FUNCTION "LAnyAxis_UnpubPhasingRelativeMasterProxy" : Void   // FC30054, SCL
TITLE = LAnyAxis_UnpubPhasingRelativeMasterProxy
{ S7_Optimized_Access := 'TRUE' }
AUTHOR : tech.team.motioncontrol@siemens.com
FAMILY : AnyAxis
VERSION : 1.0
// Support: tech.team.motioncontrol@siemens.com
   VAR_INPUT
      slave : TO_SynchronousAxis;   // Slave axis specification
      master : TO_LeadingAxisProxy;   // Master axis specification
   END_VAR
   VAR_IN_OUT
      instMC : MC_PHASINGRELATIVE;   // Instance of MC_Instruction
   END_VAR
   // Ret_Val : No return value
BEGIN
   // Call of MC_Instruction
   #instMC(Master := #master,
           Slave := #slave);
END_FUNCTION

FUNCTION "LAnyAxis_UnpubPhasingRelativeMasterSyncAxis" : Void   // FC30055, SCL
TITLE = LAnyAxis_UnpubPhasingRelativeMasterSyncAxis
{ S7_Optimized_Access := 'TRUE' }
AUTHOR : tech.team.motioncontrol@siemens.com
FAMILY : AnyAxis
VERSION : 1.0
// Support: tech.team.motioncontrol@siemens.com
   VAR_INPUT
      slave : TO_SynchronousAxis;   // Slave axis specification
      master : TO_SynchronousAxis;   // Master axis specification
   END_VAR
   VAR_IN_OUT
      instMC : MC_PHASINGRELATIVE;   // Instance of MC_Instruction
   END_VAR
   // Ret_Val : No return value
BEGIN
   // Call of MC_Instruction
   #instMC(Master := #master,
           Slave := #slave);
END_FUNCTION

// folder: LAnyAxis_Blocks/LAnyAxis_MC_TorqueData

FUNCTION_BLOCK "LAnyAxis_MC_TorqueLimiting"   // FB30042, SCL
TITLE = LAnyAxis_MC_TorqueLimiting
{ S7_Optimized_Access := 'TRUE' }
AUTHOR : tech.team.motioncontrol@siemens.com
FAMILY : AnyAxis
VERSION : 1.0
// Support: tech.team.motioncontrol@siemens.com 
// See corresponding MC_ instruction in TIA Portal help (information system)
   VAR_INPUT
      Axis : DB_ANY;   // See corresponding parameter of MC_ instruction in TIA Portal help (information system)
      Enable : Bool;   // See corresponding parameter of MC_ instruction in TIA Portal help (information system)
      Limit : LReal := -1.0;   // See corresponding parameter of MC_ instruction in TIA Portal help (information system)
      Mode : DInt;   // See corresponding parameter of MC_ instruction in TIA Portal help (information system)
   END_VAR
   VAR_OUTPUT
      InClamping : Bool;   // See corresponding parameter of MC_ instruction in TIA Portal help (information system)
      InLimitation : Bool;   // See corresponding parameter of MC_ instruction in TIA Portal help (information system)
      Busy : Bool;   // See corresponding parameter of MC_ instruction in TIA Portal help (information system)
      Error : Bool;   // See corresponding parameter of MC_ instruction in TIA Portal help (information system)
      ErrorId : Word;   // See corresponding parameter of MC_ instruction in TIA Portal help (information system)
   END_VAR
   VAR
      instMC : MC_TORQUELIMITING;   // Instance of MC_Instruction
      statEnableOld : Bool;   // Old value of execute
      statAxis : DB_ANY;   // Internal variable of axis
      statAxisType : Int;   // Actual state / axis type
   END_VAR
   VAR CONSTANT
      ERROR_INVALID_TECHNOLOGY_OBJECT : Word := 16#8002;   // See corresponding parameter of MC_ instruction in TIA Portal help (information system)
      IDLE : Int := 0;   // State idle
      INVALID_AXIS : Int := -1;   // Axis type: Invalid
      SPEED_AXIS : Int := 2;   // Axis type: Speed axis
      POSITIONING_AXIS : Int := 3;   // Axis type: Positioning axis
      SYNCHRONOUS_AXIS : Int := 4;   // Axis type: Synchronous axis
   END_VAR
BEGIN
   REGION HEADER
     //================================================================================
     // SIEMENS AG
     // (c)Copyright 2020 All Rights Reserved
     //--------------------------------------------------------------------------------
     // Library: LAnyAxis 
     // Tested with: S7-1515-2 PN
     // Engineering: TIA Portal V16
     // Restrictions: -
     // Requirements: S7-1500 FW 2.8.1
     // Functionality: Conversion DB_ANY --> TO_Axis
     // Support: tech.team.motioncontrol@siemens.com
     // Note: Parameter comments are only available in language 'English (United States)'
     //--------------------------------------------------------------------------------
     // Change log table:
     // Version  Date        Expert in charge  Changes applied
     // 01.00.00 10.03.2020  RS                First released version
     //================================================================================
   END_REGION

   REGION ENABLE
     IF (#statAxisType = #IDLE) AND #Enable THEN
       // Check axis type
       CASE TypeOfDB(#Axis) OF
         TO_POSITIONINGAXIS:
           #statAxisType := #POSITIONING_AXIS;
           #statAxis := #Axis;

         TO_SYNCHRONOUSAXIS:
           #statAxisType := #SYNCHRONOUS_AXIS;
           #statAxis := #Axis;

         TO_SPEEDAXIS:
           #statAxisType := #SPEED_AXIS;
           #statAxis := #Axis;

         ELSE
           #statAxisType := #INVALID_AXIS;
           #statAxis := 0;
       END_CASE;

     ELSIF NOT #Enable AND (#statAxisType = #INVALID_AXIS) THEN
       #statAxisType := #IDLE;

       // Outputs
       #InClamping := FALSE;
       #InLimitation := FALSE;
       #Busy := FALSE;
       #Error := FALSE;
       #ErrorId := 16#0;
     END_IF;

     // Edge detection
     #statEnableOld := #Enable;
   END_REGION

   CASE #statAxisType OF
     #IDLE:
       ;

     #POSITIONING_AXIS,
     #SYNCHRONOUS_AXIS,
     #SPEED_AXIS:
       REGION VALID_AXIS
         // Inputs
         #instMC.Enable := #Enable;
         #instMC.Limit := #Limit;
         #instMC.Mode := #Mode;

         // Call of MC instruction
         CASE #statAxisType OF
           #POSITIONING_AXIS:
             "LAnyAxis_UnpubTorqueLimitingPosAxis"(axis := #statAxis,
                                                   instMC := #instMC);
           #SYNCHRONOUS_AXIS:
             "LAnyAxis_UnpubTorqueLimitingSyncAxis"(axis := #statAxis,
                                                    instMC := #instMC);
           #SPEED_AXIS:
             #instMC(Axis := #statAxis);
         END_CASE;

         // Outputs
         #InClamping := #instMC.InClamping;
         #InLimitation := #instMC.InLimitation;
         #Busy := #instMC.Busy;
         #Error := #instMC.Error;
         #ErrorId := #instMC.ErrorId;

         // Status of MC instruction
         IF NOT #instMC.Busy
           AND NOT #instMC.Error
         THEN
           // Not active
           #statAxisType := #IDLE;
         END_IF;
       END_REGION

     ELSE
       REGION INVALID_AXIS
         // Outputs
         #InClamping := FALSE;
         #InLimitation := FALSE;
         #Busy := FALSE;
         #Error := TRUE;
         #ErrorId := #ERROR_INVALID_TECHNOLOGY_OBJECT;
       END_REGION
   END_CASE;
END_FUNCTION_BLOCK

// folder: LAnyAxis_Blocks/LAnyAxis_MC_TorqueData/InternalSubBlocks/MC_TorqueLimiting

FUNCTION "LAnyAxis_UnpubTorqueLimitingPosAxis" : Void   // FC30032, SCL
TITLE = LAnyAxis_UnpubTorqueLimitingPosAxis
{ S7_Optimized_Access := 'TRUE' }
AUTHOR : tech.team.motioncontrol@siemens.com
FAMILY : AnyAxis
VERSION : 1.0
// Support: tech.team.motioncontrol@siemens.com
   VAR_INPUT
      axis : TO_PositioningAxis;   // Axis specification
   END_VAR
   VAR_IN_OUT
      instMC : MC_TORQUELIMITING;   // Instance of MC_Instruction
   END_VAR
   // Ret_Val : No return value
BEGIN
   // Call of MC_Instruction
   #instMC(Axis := #axis);
END_FUNCTION

FUNCTION "LAnyAxis_UnpubTorqueLimitingSyncAxis" : Void   // FC30034, SCL
TITLE = LAnyAxis_UnpubTorqueLimitingSyncAxis
{ S7_Optimized_Access := 'TRUE' }
AUTHOR : tech.team.motioncontrol@siemens.com
FAMILY : AnyAxis
VERSION : 1.0
// Support: tech.team.motioncontrol@siemens.com
   VAR_INPUT
      axis : TO_SynchronousAxis;   // Axis specification
   END_VAR
   VAR_IN_OUT
      instMC : MC_TORQUELIMITING;   // Instance of MC_Instruction
   END_VAR
   // Ret_Val : No return value
BEGIN
   // Call of MC_Instruction
   #instMC(Axis := #axis);
END_FUNCTION

// folder: LAnyAxis_Blocks/LAnyAxis_TagsAccess

FUNCTION "LAnyAxis_StatusWord" : Word   // FC30077, SCL
TITLE = LAnyAxis_StatusWord
{ S7_Optimized_Access := 'TRUE' }
AUTHOR : tech.team.motioncontrol@siemens.com
FAMILY : AnyAxis
VERSION : 1.0
// Support: tech.team.motioncontrol@siemens.com
   VAR_INPUT
      axis : DB_ANY;   // Axis specification
   END_VAR
   VAR_OUTPUT
      statusWord : DWord;   // axis.StatusWord
   END_VAR
   // Ret_Val : Return value
   VAR CONSTANT
      ERROR_INVALID_TECHNOLOGY_OBJECT : Word := 16#8002;   // Error invalid TO specification
      FINISHED : Word := 16#0000;   // Finished without error
   END_VAR
BEGIN
   REGION HEADER
     //================================================================================
     // SIEMENS AG
     // (c)Copyright 2020 All Rights Reserved
     //--------------------------------------------------------------------------------
     // Library: LAnyAxis 
     // Tested with: S7-1515-2 PN
     // Engineering: TIA Portal V16
     // Restrictions: -
     // Requirements: S7-1500 FW 2.8.1
     // Functionality: Conversion DB_ANY --> TO_Axis
     // Support: tech.team.motioncontrol@siemens.com
     // Note: Parameter comments are only available in language 'English (United States)'
     //--------------------------------------------------------------------------------
     // Change log table:
     // Version  Date        Expert in charge  Changes applied
     // 01.00.00 10.03.2020  RS                First released version
     //================================================================================
   END_REGION

   // Read axis parameter
   CASE TypeOfDB(#axis) OF
     TO_POSITIONINGAXIS:
       #statusWord := "LAnyAxis_UnpubStatusWordPosAxis"(#axis);
       #LAnyAxis_StatusWord := #FINISHED;

     TO_SYNCHRONOUSAXIS:
       #statusWord := "LAnyAxis_UnpubStatusWordSyncAxis"(#axis);
       #LAnyAxis_StatusWord := #FINISHED;

     TO_EXTERNALENCODER:
       #statusWord := "LAnyAxis_UnpubStatusWordExtEncoder"(#axis);
       #LAnyAxis_StatusWord := #FINISHED;

     TO_SPEEDAXIS:
       #statusWord := "LAnyAxis_UnpubStatusWordSpeedAxis"(#axis);
       #LAnyAxis_StatusWord := #FINISHED;

     TO_LEADINGAXISPROXY:
       #statusWord := "LAnyAxis_UnpubStatusWordProxy"(#axis);
       #LAnyAxis_StatusWord := #FINISHED;

     ELSE
       #LAnyAxis_StatusWord := #ERROR_INVALID_TECHNOLOGY_OBJECT; // Invalid TO specification
   END_CASE;
END_FUNCTION

FUNCTION "LAnyAxis_StatusWord2" : Word   // FC30081, SCL
TITLE = LAnyAxis_StatusWord2
{ S7_Optimized_Access := 'TRUE' }
AUTHOR : tech.team.motioncontrol@siemens.com
FAMILY : AnyAxis
VERSION : 1.0
// Support: tech.team.motioncontrol@siemens.com
   VAR_INPUT
      axis : DB_ANY;   // Axis specification
   END_VAR
   VAR_OUTPUT
      statusWord2 : DWord;   // axis.StatusWord2
   END_VAR
   // Ret_Val : Return value
   VAR CONSTANT
      ERROR_INVALID_TECHNOLOGY_OBJECT : Word := 16#8002;   // Error invalid TO specification
      FINISHED : Word := 16#0000;   // Finished without error
   END_VAR
BEGIN
   REGION HEADER
     //================================================================================
     // SIEMENS AG
     // (c)Copyright 2020 All Rights Reserved
     //--------------------------------------------------------------------------------
     // Library: LAnyAxis 
     // Tested with: S7-1515-2 PN
     // Engineering: TIA Portal V16
     // Restrictions: -
     // Requirements: S7-1500 FW 2.8.1
     // Functionality: Conversion DB_ANY --> TO_Axis
     // Support: tech.team.motioncontrol@siemens.com
     // Note: Parameter comments are only available in language 'English (United States)'
     //--------------------------------------------------------------------------------
     // Change log table:
     // Version  Date        Expert in charge  Changes applied
     // 01.00.00 10.03.2020  RS                First released version
     //================================================================================
   END_REGION

   // Read axis parameter
   CASE TypeOfDB(#axis) OF
     TO_POSITIONINGAXIS:
       #statusWord2 := "LAnyAxis_UnpubStatusWord2PosAxis"(#axis);
       #LAnyAxis_StatusWord2 := #FINISHED;

     TO_SYNCHRONOUSAXIS:
       #statusWord2 := "LAnyAxis_UnpubStatusWord2SyncAxis"(#axis);
       #LAnyAxis_StatusWord2 := #FINISHED;

     TO_SPEEDAXIS:
       #statusWord2 := "LAnyAxis_UnpubStatusWord2SpeedAxis"(#axis);
       #LAnyAxis_StatusWord2 := #FINISHED;

     ELSE
       #LAnyAxis_StatusWord2 := #ERROR_INVALID_TECHNOLOGY_OBJECT; // Invalid TO specification
   END_CASE;
END_FUNCTION

FUNCTION "LAnyAxis_Position" : Word   // FC30087, SCL
TITLE = LAnyAxis_Position
{ S7_Optimized_Access := 'TRUE' }
AUTHOR : tech.team.motioncontrol@siemens.com
FAMILY : AnyAxis
VERSION : 1.1
// Support: tech.team.motioncontrol@siemens.com
   VAR_INPUT
      axis : DB_ANY;   // Axis specification
   END_VAR
   VAR_OUTPUT
      position : LReal;   // axis.Position
   END_VAR
   // Ret_Val : Return value
   VAR CONSTANT
      ERROR_INVALID_TECHNOLOGY_OBJECT : Word := 16#8002;   // Error invalid TO specification
      FINISHED : Word := 16#0000;   // Finished without error
   END_VAR
BEGIN
   REGION HEADER
     //================================================================================
     // SIEMENS AG
     // (c)Copyright 2021 All Rights Reserved
     //--------------------------------------------------------------------------------
     // Library: LAnyAxis 
     // Tested with: S7-1515-2 PN
     // Engineering: TIA Portal V17
     // Restrictions: -
     // Requirements: S7-1500 FW 2.9
     // Functionality: Conversion DB_ANY --> TO_Axis
     // Support: tech.team.motioncontrol@siemens.com
     // Note: Parameter comments are only available in language 'English (United States)'
     //--------------------------------------------------------------------------------
     // Change log table:
     // Version  Date        Expert in charge  Changes applied
     // 01.00.00 01.01.2021  RS                First released version
     // 01.01.00 24.02.2021  RS                Update MC V6.0
     //================================================================================
   END_REGION

   // Read axis parameter
   CASE TypeOfDB(#axis) OF
     TO_POSITIONINGAXIS:
       #position := "LAnyAxis_UnpubPositionPosAxis"(#axis);
       #LAnyAxis_Position := #FINISHED;

     TO_SYNCHRONOUSAXIS:
       #position := "LAnyAxis_UnpubPositionSyncAxis"(#axis);
       #LAnyAxis_Position := #FINISHED;

     TO_LEADINGAXISPROXY:
       #position := "LAnyAxis_UnpubPositionProxy"(#axis);
       #LAnyAxis_Position := #FINISHED;

     ELSE
       #LAnyAxis_Position := #ERROR_INVALID_TECHNOLOGY_OBJECT; // Invalid TO specification
   END_CASE;
END_FUNCTION

// folder: LAnyAxis_Blocks/LAnyAxis_TagsAccess/InternalSubBlocks/Position

FUNCTION "LAnyAxis_UnpubPositionPosAxis" : LReal   // FC30085, SCL
TITLE = LAnyAxis_UnpubPositionPosAxis
{ S7_Optimized_Access := 'TRUE' }
AUTHOR : tech.team.motioncontrol@siemens.com
FAMILY : AnyAxis
VERSION : 1.0
// Support: tech.team.motioncontrol@siemens.com
   VAR_INPUT
      axis : TO_PositioningAxis;   // Axis specification
   END_VAR
   // Ret_Val : axis.Position
BEGIN
   // Read axis parameter
   #LAnyAxis_UnpubPositionPosAxis := #axis.Position;
END_FUNCTION

FUNCTION "LAnyAxis_UnpubPositionSyncAxis" : LReal   // FC30086, SCL
TITLE = LAnyAxis_UnpubPositionSyncAxis
{ S7_Optimized_Access := 'TRUE' }
AUTHOR : tech.team.motioncontrol@siemens.com
FAMILY : AnyAxis
VERSION : 1.0
// Support: tech.team.motioncontrol@siemens.com
   VAR_INPUT
      axis : TO_SynchronousAxis;   // Axis specification
   END_VAR
   // Ret_Val : axis.Position
BEGIN
   // Read axis parameter
   #LAnyAxis_UnpubPositionSyncAxis := #axis.Position;
END_FUNCTION

FUNCTION "LAnyAxis_UnpubPositionProxy" : LReal   // FC30139, SCL
TITLE = LAnyAxis_UnpubPositionProxy
{ S7_Optimized_Access := 'TRUE' }
AUTHOR : tech.team.motioncontrol@siemens.com
FAMILY : AnyAxis
VERSION : 1.0
// Support: tech.team.motioncontrol@siemens.com
   VAR_INPUT
      axis : TO_LeadingAxisProxy;   // Axis specification
   END_VAR
   // Ret_Val : axis.Position
BEGIN
   // Read axis parameter
   #LAnyAxis_UnpubPositionProxy := #axis.Position;
END_FUNCTION

// folder: LAnyAxis_Blocks/LAnyAxis_TagsAccess/InternalSubBlocks/StatusWord

FUNCTION "LAnyAxis_UnpubStatusWordExtEncoder" : DWord   // FC30073, SCL
TITLE = LAnyAxis_UnpubStatusWordExtEncoder
{ S7_Optimized_Access := 'TRUE' }
AUTHOR : tech.team.motioncontrol@siemens.com
FAMILY : AnyAxis
VERSION : 1.0
// Support: tech.team.motioncontrol@siemens.com
   VAR_INPUT
      axis : TO_ExternalEncoder;   // Axis specification
   END_VAR
   // Ret_Val : axis.StatusWord
BEGIN
   // Read axis parameter
   #LAnyAxis_UnpubStatusWordExtEncoder := #axis.StatusWord;
END_FUNCTION

FUNCTION "LAnyAxis_UnpubStatusWordPosAxis" : DWord   // FC30074, SCL
TITLE = LAnyAxis_UnpubStatusWordPosAxis
{ S7_Optimized_Access := 'TRUE' }
AUTHOR : tech.team.motioncontrol@siemens.com
FAMILY : AnyAxis
VERSION : 1.0
// Support: tech.team.motioncontrol@siemens.com
   VAR_INPUT
      axis : TO_PositioningAxis;   // Axis specification
   END_VAR
   // Ret_Val : axis.StatusWord
BEGIN
   // Read axis parameter
   #LAnyAxis_UnpubStatusWordPosAxis := #axis.StatusWord;
END_FUNCTION

FUNCTION "LAnyAxis_UnpubStatusWordProxy" : DWord   // FC30075, SCL
TITLE = LAnyAxis_UnpubStatusWordProxy
{ S7_Optimized_Access := 'TRUE' }
AUTHOR : tech.team.motioncontrol@siemens.com
FAMILY : AnyAxis
VERSION : 1.0
// Support: tech.team.motioncontrol@siemens.com
   VAR_INPUT
      axis : TO_LeadingAxisProxy;   // Axis specification
   END_VAR
   // Ret_Val : axis.StatusWord
BEGIN
   // Read axis parameter
   #LAnyAxis_UnpubStatusWordProxy := #axis.StatusWord;
END_FUNCTION

FUNCTION "LAnyAxis_UnpubStatusWordSyncAxis" : DWord   // FC30076, SCL
TITLE = LAnyAxis_UnpubStatusWordSyncAxis
{ S7_Optimized_Access := 'TRUE' }
AUTHOR : tech.team.motioncontrol@siemens.com
FAMILY : AnyAxis
VERSION : 1.0
// Support: tech.team.motioncontrol@siemens.com
   VAR_INPUT
      axis : TO_SynchronousAxis;   // Axis specification
   END_VAR
   // Ret_Val : axis.StatusWord
BEGIN
   // Read axis parameter
   #LAnyAxis_UnpubStatusWordSyncAxis := #axis.StatusWord;
END_FUNCTION

FUNCTION "LAnyAxis_UnpubStatusWordSpeedAxis" : DWord   // FC30079, SCL
TITLE = LAnyAxis_UnpubStatusWordSpeedAxis
{ S7_Optimized_Access := 'TRUE' }
AUTHOR : tech.team.motioncontrol@siemens.com
FAMILY : AnyAxis
VERSION : 1.0
// Support: tech.team.motioncontrol@siemens.com
   VAR_INPUT
      axis : TO_SpeedAxis;   // Axis specification
   END_VAR
   // Ret_Val : axis.StatusWord
BEGIN
   // Read axis parameter
   #LAnyAxis_UnpubStatusWordSpeedAxis := #axis.StatusWord;
END_FUNCTION

// folder: LAnyAxis_Blocks/LAnyAxis_TagsAccess/InternalSubBlocks/StatusWord2

FUNCTION "LAnyAxis_UnpubStatusWord2SpeedAxis" : DWord   // FC30072, SCL
TITLE = LAnyAxis_UnpubStatusWordSpeedAxis
{ S7_Optimized_Access := 'TRUE' }
AUTHOR : tech.team.motioncontrol@siemens.com
FAMILY : AnyAxis
VERSION : 1.0
// Support: tech.team.motioncontrol@siemens.com
   VAR_INPUT
      axis : TO_SpeedAxis;   // Axis specification
   END_VAR
   // Ret_Val : axis.StatusWord2
BEGIN
   // Read axis parameter
   #LAnyAxis_UnpubStatusWord2SpeedAxis := #axis.StatusWord2;
END_FUNCTION

FUNCTION "LAnyAxis_UnpubStatusWord2PosAxis" : DWord   // FC30078, SCL
TITLE = LAnyAxis_UnpubStatusWord2PosAxis
{ S7_Optimized_Access := 'TRUE' }
AUTHOR : tech.team.motioncontrol@siemens.com
FAMILY : AnyAxis
VERSION : 1.0
// Support: tech.team.motioncontrol@siemens.com
   VAR_INPUT
      axis : TO_PositioningAxis;   // Axis specification
   END_VAR
   // Ret_Val : axis.StatusWord2
BEGIN
   // Read axis parameter
   #LAnyAxis_UnpubStatusWord2PosAxis := #axis.StatusWord2;
END_FUNCTION

FUNCTION "LAnyAxis_UnpubStatusWord2SyncAxis" : DWord   // FC30080, SCL
TITLE = LAnyAxis_UnpubStatusWord2SyncAxis
{ S7_Optimized_Access := 'TRUE' }
AUTHOR : tech.team.motioncontrol@siemens.com
FAMILY : AnyAxis
VERSION : 1.0
// Support: tech.team.motioncontrol@siemens.com
   VAR_INPUT
      axis : TO_SynchronousAxis;   // Axis specification
   END_VAR
   // Ret_Val : axis.StatusWord2
BEGIN
   // Read axis parameter
   #LAnyAxis_UnpubStatusWord2SyncAxis := #axis.StatusWord2;
END_FUNCTION

// folder: LAnyAxis_Blocks/LAnyAxis_TagsAccess/Modulo

FUNCTION "LAnyAxis_ModuloEnable" : Word   // FC30114, SCL
TITLE = LAnyAxis_ModuloEnable
{ S7_Optimized_Access := 'TRUE' }
AUTHOR : tech.team.motioncontrol@siemens.com
FAMILY : AnyAxis
VERSION : 1.1
// Support: tech.team.motioncontrol@siemens.com
   VAR_INPUT
      axis : DB_ANY;   // Axis specification
   END_VAR
   VAR_OUTPUT
      enable : Bool;   // axis.Modulo.Enable
   END_VAR
   // Ret_Val : Return value
   VAR CONSTANT
      ERROR_INVALID_TECHNOLOGY_OBJECT : Word := 16#8002;   // Error invalid TO specification
      FINISHED : Word := 16#0000;   // Finished without error
   END_VAR
BEGIN
   REGION HEADER
     //================================================================================
     // SIEMENS AG
     // (c)Copyright 2021 All Rights Reserved
     //--------------------------------------------------------------------------------
     // Library: LAnyAxis 
     // Tested with: S7-1515-2 PN
     // Engineering: TIA Portal V17
     // Restrictions: -
     // Requirements: S7-1500 FW 2.9
     // Functionality: Conversion DB_ANY --> TO_Axis
     // Support: tech.team.motioncontrol@siemens.com
     // Note: Parameter comments are only available in language 'English (United States)'
     //--------------------------------------------------------------------------------
     // Change log table:
     // Version  Date        Expert in charge  Changes applied
     // 01.00.00 01.01.2021  RS                First released version
     // 01.01.00 24.02.2021  RS                Update MC V6.0
     //================================================================================
   END_REGION

   // Read axis parameter
   CASE TypeOfDB(#axis) OF
     TO_POSITIONINGAXIS:
       #enable := "LAnyAxis_UnpubModuloEnablePosAxis"(#axis);
       #LAnyAxis_ModuloEnable := #FINISHED;

     TO_SYNCHRONOUSAXIS:
       #enable := "LAnyAxis_UnpubModuloEnableSyncAxis"(#axis);
       #LAnyAxis_ModuloEnable := #FINISHED;

     TO_EXTERNALENCODER:
       #enable := "LAnyAxis_UnpubModuloEnableExtEncoder"(#axis);
       #LAnyAxis_ModuloEnable := #FINISHED;

     ELSE
       #LAnyAxis_ModuloEnable := #ERROR_INVALID_TECHNOLOGY_OBJECT; // Invalid TO specification
   END_CASE;
END_FUNCTION

// folder: LAnyAxis_Blocks/LAnyAxis_TagsAccess/Modulo/InternalSubBlocks/Enable

FUNCTION "LAnyAxis_UnpubModuloEnableExtEncoder" : Bool   // FC30093, SCL
TITLE = LAnyAxis_UnpubModuloEnableExtEncoder
{ S7_Optimized_Access := 'TRUE' }
AUTHOR : tech.team.motioncontrol@siemens.com
FAMILY : AnyAxis
VERSION : 1.0
// Support: tech.team.motioncontrol@siemens.com
   VAR_INPUT
      axis : TO_ExternalEncoder;   // Axis specification
   END_VAR
   // Ret_Val : axis.Modulo.Enable
BEGIN
   // Read axis parameter
   #LAnyAxis_UnpubModuloEnableExtEncoder := #axis.Modulo.Enable;
END_FUNCTION

FUNCTION "LAnyAxis_UnpubModuloEnablePosAxis" : Bool   // FC30094, SCL
TITLE = LAnyAxis_UnpubModuloEnablePosAxis
{ S7_Optimized_Access := 'TRUE' }
AUTHOR : tech.team.motioncontrol@siemens.com
FAMILY : AnyAxis
VERSION : 1.0
// Support: tech.team.motioncontrol@siemens.com
   VAR_INPUT
      axis : TO_PositioningAxis;   // Axis specification
   END_VAR
   // Ret_Val : axis.Modulo.Enable
BEGIN
   // Read axis parameter
   #LAnyAxis_UnpubModuloEnablePosAxis := #axis.Modulo.Enable;
END_FUNCTION

FUNCTION "LAnyAxis_UnpubModuloEnableSyncAxis" : Bool   // FC30095, SCL
TITLE = LAnyAxis_UnpubModuloEnableSyncAxis
{ S7_Optimized_Access := 'TRUE' }
AUTHOR : tech.team.motioncontrol@siemens.com
FAMILY : AnyAxis
VERSION : 1.0
// Support: tech.team.motioncontrol@siemens.com
   VAR_INPUT
      axis : TO_SynchronousAxis;   // Axis specification
   END_VAR
   // Ret_Val : axis.Modulo.Enable
BEGIN
   // Read axis parameter
   #LAnyAxis_UnpubModuloEnableSyncAxis := #axis.Modulo.Enable;
END_FUNCTION

// ===== library: MasterCopy "LAxisCtrl_typeCamIn" =====

// folder: LAxisCtrl_Types/LAxisCtrl_SubTypes

TYPE "LAxisCtrl_typeCamIn"
TITLE = LAxisCtrl_typeCamIn
// Support: tech.team.motioncontrol@siemens.com
   STRUCT
      masterOffset : LReal := 0.0;   // Offset of leading values of cam
      slaveOffset : LReal := 0.0;   // Offset of following values of cam
      masterScaling : LReal := 1.0;   // Scaling the leading values of the cam
      slaveScaling : LReal := 1.0;   // Scaling the following values of the cam
      masterSyncPosition : LReal := 0.0;   // Starting point in the cam/distance from the cam start with reference to the scaled cam
      syncProfileReference : DInt := 1;   // Synchronization profile (0: Synchronization in advance using dynamic parameters; 1: Synchronization in advance using leading value distance; 2: Direct synchronous setting; 3: Subsequent synchronization using leading value distance; 4: Subsequent synchronization using leading value distance starting from current leading value position; 5: Direct synchronous setting at the end of the cam)
      masterStartDistance : LReal := 0.0;   // Leading value distance when "SyncProfileReference" = 1, 3, 4
      velocity : LReal := -1.0;   // Velocity for synchronization (Value > 0.0: The specified value is used; Value = 0.0: Not permitted; Value < 0.0: Use of the default value configured in the technology object) when "SyncProfileReference" = 0
      acceleration : LReal := -1.0;   // Acceleration for synchronization (Value > 0.0: The specified value is used; Value = 0.0: Not permitted; Value < 0.0: Use of the default value configured in the technology object) when "SyncProfileReference" = 0
      deceleration : LReal := -1.0;   // Deceleration for synchronization (Value > 0.0: The specified value is used; Value = 0.0: Not permitted; Value < 0.0: Use of the default value configured in the technology object) when "SyncProfileReference" = 0
      jerk : LReal := -1.0;   // Jerk for synchronization (Value > 0.0: Smooth velocity profile, the specified value is used; Value = 0.0: Trapezoid velocity profile; Value < 0.0: Use of the default value configured in the technology object) when "SyncProfileReference" = 0
      applicationMode : DInt := 0;   // Application of the cam (0: Once/not cyclic; 1: Cyclic (absolute application on the following value side); 2: Cyclic appending (continuously appending on the following value side))
      syncDirection : DInt := 1;   // Direction for synchronization only in effect for axes with activated modulo setting (1: Forward direction; 2: Backward direction; 3: Shortest way) when "SyncProfileReference" = 0, 1, 3, 4
   END_STRUCT;
END_TYPE

// ===== library: MasterCopy "LAxisCtrl_typeFastStop" =====

// folder: LAxisCtrl_Types/LAxisCtrl_SubTypes

TYPE "LAxisCtrl_typeFastStop"
TITLE = LAxisCtrl_typeFastStop
// Support: tech.team.motioncontrol@siemens.com
   STRUCT
      deceleration : LReal := -1.0;   // Deceleration for fast stop (Value > 0.0: The specified value is used; Value <= 0.0: Emergency deceleration of the technology object is used)
      jerk : LReal := -1.0;   // Jerk for fast stop (Value > 0.0: Smooth velocity profile, the specified value is used; Value = 0.0: Trapezoid velocity profile; Value < 0.0: Use of the default value configured in the technology object)
      abortAcceleration : Bool := FALSE;   // TRUE: The acceleration is set to 0.0 at the start of the job, and the deceleration immediately builds up; FALSE: The current acceleration at the start of the job is reduced using the configured jerk. Afterwards, the deceleration builds up
      replaceStopPossible : Bool := FALSE;   // TRUE: Fast stop command can be replaced by another command
   END_STRUCT;
END_TYPE

// ===== library: MasterCopy "LAxisCtrl_typeGearInAbsolute" =====

// folder: LAxisCtrl_Types/LAxisCtrl_SubTypes

TYPE "LAxisCtrl_typeGearInAbsolute"
TITLE = LAxisCtrl_typeGearInAbsolute
// Support: tech.team.motioncontrol@siemens.com
   STRUCT
      ratioNumerator : DInt := 1;   // Gear ratio numerator (permitted integer values: -2147483648 to 2147483647; value 0 not permitted)
      ratioDenominator : DInt := 1;   // Gear ratio denominator (permitted integer values: 1 to 2147483647)
      masterSyncPosition : LReal := 0.0;   // Synchronous position of leading axis
      slaveSyncPosition : LReal := 0.0;   // Synchronous position of following axis
      syncProfileReference : DInt := 1;   // Type of synchronization (0: Synchronization in advance using dynamic parameters; 1: Synchronization in advance using leading value distance; 3: Subsequent synchronization using leading value distance)
      masterStartDistance : LReal := 0.0;   // Leading value distance when "SyncProfileReference" = 1, 3
      velocity : LReal := -1.0;   // Velocity for synchronization (Value > 0.0: The specified value is used; Value = 0.0: Not permitted; Value < 0.0: Use of the default value configured in the technology object) when "SyncProfileReference" = 0
      acceleration : LReal := -1.0;   // Acceleration for synchronization (Value > 0.0: The specified value is used; Value = 0.0: Not permitted; Value < 0.0: Use of the default value configured in the technology object) when "SyncProfileReference" = 0
      deceleration : LReal := -1.0;   // Deceleration for synchronization (Value > 0.0: The specified value is used; Value = 0.0: Not permitted; Value < 0.0: Use of the default value configured in the technology object) when "SyncProfileReference" = 0
      jerk : LReal := -1.0;   // Jerk for synchronization (Value > 0.0: Smooth velocity profile, the specified value is used; Value = 0.0: Trapezoid velocity profile; Value < 0.0: Use of the default value configured in the technology object) when "SyncProfileReference" = 0
      syncDirection : DInt := 1;   // Direction for synchronization only in effect for axes with activated modulo setting (1: Forward direction; 2: Backward direction; 3: Shortest way)
      ratioChangeOnTheFly : Bool := FALSE;   // TRUE: Changing gear ratio on-the-fly; FALSE: Ratio change requires a new rising edge at gearInAbsolute input
   END_STRUCT;
END_TYPE

// ===== library: MasterCopy "LAxisCtrl_typeGeneralSettings" =====

// folder: LAxisCtrl_Types/LAxisCtrl_SubTypes

TYPE "LAxisCtrl_typeGeneralSettings"
TITLE = LAxisCtrl_typeGeneralSettings
// Support: tech.team.motioncontrol@siemens.com
   STRUCT
      stopOnError : Bool := TRUE;   // TRUE: In case of error the axis will be stopped automatically with fastStop dynamics
      resetWithRestart : Bool := FALSE;   // TRUE: Reinitialization of the technology object and acknowledgment of pending technology alarms. The technology object is reinitialized with the configured start values; FALSE: Acknowledgment of queued technology alarms
      abortWaitingSyncCmd : Bool := TRUE;   // TRUE: Abort waiting synchronous command (MC_GEARINPOS, MC_CAMIN) in case of new basic motion command automatically
   END_STRUCT;
END_TYPE

// ===== library: MasterCopy "LAxisCtrl_typeHoming" =====

// folder: LAxisCtrl_Types/LAxisCtrl_SubTypes

TYPE "LAxisCtrl_typeHoming"
TITLE = LAxisCtrl_typeHoming
// Support: tech.team.motioncontrol@siemens.com
   STRUCT
      position : LReal := 0.0;   // The specified value is used according to the selected "Mode"
      mode : Int := 0;   // Operation mode; 0: Direct homing (absolute); 1: Direct homing (relative); 2: Passive homing (without reset); 3: Active homing; 5: Active homing (Position parameter has no effect); 6: Absolute encoder adjustment (relative); 7: Absolute encoder adjustment (absolute); 8: Passive homing; 9: Abort passive homing; 10: Passive homing (Position parameter has no effect); 11: Set setpoint position (absolute); 12: Shift the setpoint position (relative)
      extendedMode : DInt := -1;   // -1: No extended homing mode (parameter "mode" is effective); 0: Homing on fixed stop; 1: Homing on fixed stop with moving out of clamping; 2: Homing on fixed stop with moving to target position
      extendedModeTorqueLimit : LReal := 0.0;   // Value of the torque/force for extended homing mode
      extendedModeTargetPosition : LReal := 0.0;   // Target position when 'extendedMode' = 2
   END_STRUCT;
END_TYPE

// ===== library: MasterCopy "LAxisCtrl_typeJog" =====

// folder: LAxisCtrl_Types/LAxisCtrl_SubTypes

TYPE "LAxisCtrl_typeJog"
TITLE = LAxisCtrl_typeJog
// Support: tech.team.motioncontrol@siemens.com
   STRUCT
      velocity : LReal := 0.0;   // Velocity for jogging (Value > 0.0: The specified value is used; Value = 0.0: Permitted; Value < 0.0: The absolute value of the specified value is used)
      acceleration : LReal := -1.0;   // Acceleration for jogging (Value > 0.0: The specified value is used; Value = 0.0: Not permitted; Value < 0.0: Use of the default value configured in the technology object)
      deceleration : LReal := -1.0;   // Deceleration for jogging (Value > 0.0: The specified value is used; Value = 0.0: Not permitted; Value < 0.0: Use of the default value configured in the technology object)
      jerk : LReal := -1.0;   // Jerk for jogging (Value > 0.0: Smooth velocity profile, the specified value is used; Value = 0.0: Trapezoid velocity profile; Value < 0.0: Use of the default value configured in the technology object)
      positionControlled : Bool := TRUE;   // TRUE: Position-controlled mode; FALSE: Non position-controlled operation
      increment : LReal := 0.0;   // Increment/distance for incremental jogging
      mode : DInt := 0;   // 0: Continuous jogging; 1: Incremental jogging new increment (starts with new increment); 2: Incremental jogging continue increment (continue the last increment if not completed)
   END_STRUCT;
END_TYPE

// ===== library: MasterCopy "LAxisCtrl_typeMoveVelocity" =====

// folder: LAxisCtrl_Types/LAxisCtrl_SubTypes

TYPE "LAxisCtrl_typeMoveVelocity"
TITLE = LAxisCtrl_typeMoveVelocity
// Support: tech.team.motioncontrol@siemens.com
   STRUCT
      velocity : LReal := 0.0;   // Velocity/Speed for motion process (Value = 0.0: Permitted)
      acceleration : LReal := -1.0;   // Acceleration setpoint for motion process (Value > 0.0: The specified value is used; Value = 0.0: Not permitted; Value < 0.0: Use of the default value configured in the technology object)
      deceleration : LReal := -1.0;   // Deceleration setpoint for motion process (Value > 0.0: The specified value is used; Value = 0.0: Not permitted; Value < 0.0: Use of the default value configured in the technology object)
      jerk : LReal := -1.0;   // Jerk for velocity specification (Value > 0.0: Smooth velocity profile, the specified value is used; (Value = 0.0: Trapezoid velocity profile; (Value < 0.0: Use of the default value configured in the technology object)
      direction : Int := 0;   // Motion direction of the axis (0: The sign of the velocity parameter defines the direction; 1: Positive direction; 2: Negative direction)
      positionControlled : Bool := TRUE;   // TRUE: Position-controlled operation; FALSE: Non position-controlled operation
      velocityChangeOnTheFly : Bool := FALSE;   // TRUE: Changing velocity on-the-fly; FALSE: Velocity change requires a new rising edge on moveVelocity input
   END_STRUCT;
END_TYPE

// ===== library: MasterCopy "LAxisCtrl_typeOffset" =====

// folder: LAxisCtrl_Types/LAxisCtrl_SubTypes

TYPE "LAxisCtrl_typeOffset"
TITLE = LAxisCtrl_typeOffset
// Support: tech.team.motioncontrol@siemens.com
   STRUCT
      offset : LReal := 0.0;   // Absolute or relative offset shift
      profileReference : DInt := 1;   // Type of traversing of the following value offset (1: Traverse following value offset using leading value distance starting from the current effective leading value position; 2: Traverse following value offset using leading value distance from the effective leading value position "StartPosition"; 5: Cancel only one waiting job for the following value offset)
      offsetDistance : LReal;   // Effective leading value distance while traversing the following value offset when "ProfileReference" = 1, 2
      startPosition : LReal;   // Effective leading value position starting from which the following value offset is traversed when "ProfileReference" = 2
      direction : DInt := 3;   // Direction of the leading value distance (1: Positive direction; 2: Negative direction; 3: Current direction) when "ProfileReference" = 1, 2
      offsetAbsolute : Bool := TRUE;   // Indicates the type of the offset shift. TRUE: Shift the following value as an absolute shift; FALSE: Shift the following value relative to the existing following value shift
      offsetChangeOnTheFly : Bool := FALSE;   // TRUE: Changing offset shift on-the-fly at absolute offset shift. FALSE: Offset shift change requires a new rising edge at offset input
   END_STRUCT;
END_TYPE

// ===== library: MasterCopy "LAxisCtrl_typePhasing" =====

// folder: LAxisCtrl_Types/LAxisCtrl_SubTypes

TYPE "LAxisCtrl_typePhasing"
TITLE = LAxisCtrl_typePhasing
// Support: tech.team.motioncontrol@siemens.com
   STRUCT
      phaseShift : LReal := 0.0;   // Absolute or relative leading value shift
      velocity : LReal := -1.0;   // Velocity for leading value shift, added to synchronous operation motion (Value > 0.0: The specified value is used; Value = 0.0: Not permitted; Value < 0.0: Use of the default value configured in the technology object)
      acceleration : LReal := -1.0;   // Acceleration for leading value shift, added to synchronous operation motion (Value > 0.0: The specified value is used; Value = 0.0: Not permitted; Value < 0.0: Use of the default value configured in the technology object)
      deceleration : LReal := -1.0;   // Deceleration for leading value shift, added to synchronous operation motion (Value > 0.0: The specified value is used; Value = 0.0: Not permitted; Value < 0.0: Use of the default value configured in the technology object)
      jerk : LReal := -1.0;   // Jerk for leading value shift, added to synchronous operation motion (Value > 0.0: Smooth velocity profile, the specified value is used; Value = 0.0: Trapezoid velocity profile; Value < 0.0: Use of the default value configured in the technology object)
      profileReference : DInt;   // Type of traversing of the leading value offset (0: Only with gearing: Traverse leading value offset using dynamics parameters; 1: Traverse leading value offset via leading value distance starting from current leading value position; 2: Traverse leading value offset from leading value position "StartPosition"; 5: Cancel only one waiting job for the leading value offset)
      phasingDistance : LReal;   // Leading value distance (Distance of the leading axis during the traversing of the leading value offset) when "ProfileReference" = 1, 2
      startPosition : LReal;   // Leading value position starting from which the leading value offset is traversed when "ProfileReference" = 2
      direction : DInt := 3;   // Direction of the leading value distance (1: Positive direction; 2: Negative direction; 3: Current direction) when "ProfileReference" = 1, 2
      phaseAbsolute : Bool := TRUE;   // Indicates the type of phase shift. TRUE: Shift the leading value as an absolute shift; FALSE: Shift the leading value relative to the existing leading value shift
      phaseShiftChangeOnTheFly : Bool := FALSE;   // TRUE: Changing phase shift on-the-fly at absolute phasing; FALSE: Phase shift change requires a new rising edge at phasing input
   END_STRUCT;
END_TYPE

// ===== library: MasterCopy "LAxisCtrl_typePosAbsolute" =====

// folder: LAxisCtrl_Types/LAxisCtrl_SubTypes

TYPE "LAxisCtrl_typePosAbsolute"
TITLE = LAxisCtrl_typePosAbsolute
// Support: tech.team.motioncontrol@siemens.com
   STRUCT
      position : LReal := 0.0;   // Absolute target position
      velocity : LReal := -1.0;   // Velocity setpoint for absolute positioning (Value > 0.0: The specified value is used; Value = 0.0: Not permitted; Value < 0.0: Use of the default value configured in the technology object)
      acceleration : LReal := -1.0;   // Acceleration setpoint for absolute positioning (Value > 0.0: The specified value is used; Value = 0.0: Not permitted; Value < 0.0: Use of the default value configured in the technology object)
      deceleration : LReal := -1.0;   // Deceleration setpoint for absolute positioning (Value > 0.0: The specified value is used; Value = 0.0: Not permitted; Value < 0.0: Use of the default value configured in the technology object)
      jerk : LReal := -1.0;   // Jerk for absolute positioning (Value > 0.0: Smooth velocity profile, the specified value is used; (Value = 0.0: Trapezoid velocity profile; (Value < 0.0: Use of the default value configured in the technology object)
      direction : Int := 1;   // Motion direction of the axis (1: Positive direction; 2: Negative direction; 3: Shortest way)
      positionChangeOnTheFly : Bool := FALSE;   // TRUE: Changing position on-the-fly; FALSE: Position change requires a new rising edge at posAbsolute input
      velocityChangeOnTheFly : Bool := FALSE;   // TRUE: Changing velocity on-the-fly; FALSE: Velocity change requires a new rising edge at posAbsolute input
   END_STRUCT;
END_TYPE

// ===== library: MasterCopy "LAxisCtrl_typePosRelative" =====

// folder: LAxisCtrl_Types/LAxisCtrl_SubTypes

TYPE "LAxisCtrl_typePosRelative"
TITLE = LAxisCtrl_typePosRelative
// Support: tech.team.motioncontrol@siemens.com
   STRUCT
      distance : LReal := 0.0;   // Distance for positioning process
      velocity : LReal := -1.0;   // Velocity setpoint for relative positioning (Value > 0.0: The specified value is used; Value = 0.0: Not permitted; Value < 0.0: Use of the default value configured in the technology object)
      acceleration : LReal := -1.0;   // Acceleration setpoint for relative positioning (Value > 0.0: The specified value is used; Value = 0.0: Not permitted; Value < 0.0: Use of the default value configured in the technology object)
      deceleration : LReal := -1.0;   // Deceleration setpoint for relative positioning (Value > 0.0: The specified value is used; Value = 0.0: Not permitted; Value < 0.0: Use of the default value configured in the technology object)
      jerk : LReal := -1.0;   // Jerk for relative positioning (Value > 0.0: Smooth velocity profile, the specified value is used; Value = 0.0: Trapezoid velocity profile; Value < 0.0: Use of the default value configured in the technology object)
      direction : DInt := 0;   // Motion direction of the axis (0: The sign of the distance parameter defines the direction; 1: Positive direction; 2: Negative direction)
   END_STRUCT;
END_TYPE

// ===== library: MasterCopy "LAxisCtrl_typePosSuperimposed" =====

// folder: LAxisCtrl_Types/LAxisCtrl_SubTypes

TYPE "LAxisCtrl_typePosSuperimposed"
TITLE = LAxisCtrl_typePosSuperimposed
// Support: tech.team.motioncontrol@siemens.com
   STRUCT
      distance : LReal := 0.0;   // Distance for superimposed positioning
      velocityDiff : LReal := -1.0;   // Maximum velocity deviation compared to the active motion (Value > 0.0: The specified value is used; Value = 0.0: Not permitted; Value < 0.0: Use of the default value configured in the technology object)
      acceleration : LReal := -1.0;   // Acceleration for positioning (Value > 0.0: The specified value is used; Value = 0.0: Not permitted; Value < 0.0: Use of the default value configured in the technology object)
      deceleration : LReal := -1.0;   // Deceleration for positioning (Value > 0.0: The specified value is used; Value = 0.0: Not permitted; Value < 0.0: Use of the default value configured in the technology object)
      jerk : LReal := -1.0;   // Jerk for positioning (Value > 0.0: Smooth velocity profile, the specified value is used; Value = 0.0: Trapezoid velocity profile; Value < 0.0: Use of the default value configured in the technology object)
      direction : DInt := 0;   // Motion direction of the axis (0: The sign of the distance parameter defines the direction; 1: Positive negative; 2: Negative direction)
   END_STRUCT;
END_TYPE

// ===== library: MasterCopy "LAxisCtrl_typePower" =====

// folder: LAxisCtrl_Types/LAxisCtrl_SubTypes

TYPE "LAxisCtrl_typePower"
TITLE = LAxisCtrl_typePower
// Support: tech.team.motioncontrol@siemens.com
   STRUCT
      startMode : DInt := 1;   // 0: Enable axis not position-controlled; 1: Enable axis position-controlled (This parameter is ignored when a speed axis or external encoder is used)
      stopMode : Int := 0;   // 0: Emergency stop; 1: Immediate stop; 2: Stop with maximum dynamic values
      syncMotionSimulation : Bool := FALSE;   // TRUE: Start the simulation of synchronous operation automatically with falling edge at enableAxis; FALSE: No simulation of synchronous operation
      syncMotionSimulationExtendedMode : Int := -1;   // Only valid if 'syncMotionSimulation' = TRUE: -1: Start the simulation of synchronous operation only if the axis is in synchronous operation; 0: Start the simulation of synchronous operation independently from the synchronous operation state
   END_STRUCT;
END_TYPE

// ===== library: MasterCopy "LAxisCtrl_typeStop" =====

// folder: LAxisCtrl_Types/LAxisCtrl_SubTypes

TYPE "LAxisCtrl_typeStop"
TITLE = LAxisCtrl_typeStop
// Support: tech.team.motioncontrol@siemens.com
   STRUCT
      deceleration : LReal := -1.0;   // Deceleration setpoint for stop (Value > 0.0: The specified value is used; Value = 0.0: Not permitted; Value < 0.0: Use of the default value configured in the technology object)
      jerk : LReal := -1.0;   // Jerk for stop (Value > 0.0: Smooth velocity profile, the specified value is used; Value = 0.0: Trapezoid velocity profile; Value < 0.0: Use of the default value configured in the technology object)
      abortAcceleration : Bool := FALSE;   // TRUE: The acceleration is set to 0.0 at the start of the job, and the deceleration immediately builds up; FALSE: The current acceleration at the start of the job is reduced using the configured jerk. Afterwards, the deceleration builds up
   END_STRUCT;
END_TYPE

// ===== library: MasterCopy "LAxisCtrl_typeTorqueLimiting" =====

// folder: LAxisCtrl_Types/LAxisCtrl_SubTypes

TYPE "LAxisCtrl_typeTorqueLimiting"
TITLE = LAxisCtrl_typeTorqueLimiting
// Support: tech.team.motioncontrol@siemens.com
   STRUCT
      limit : LReal := -1.0;   // Value of force/torque limiting (in the configured unit of measurement) (Value >= 0.0: The specified value is used; Value < 0.0: Use of the default value configured in the technology object)
      mode : DInt := 0;   // 0: Force/Torque limiting; 1: Fixed stop detection
   END_STRUCT;
END_TYPE

// ===== library: MasterCopy "LAxisCtrl_typeAxisConfig" =====

// folder: LAxisCtrl_Types

TYPE "LAxisCtrl_typeAxisConfig"
TITLE = LAxisCtrl_typeAxisConfig
// Support: tech.team.motioncontrol@siemens.com
   STRUCT
      generalSettings : "LAxisCtrl_typeGeneralSettings";   // Configuration of general settings
      power : "LAxisCtrl_typePower";   // Configuration of MC_POWER function
      jog : "LAxisCtrl_typeJog";   // Configuration of JOG function
      moveVelocity : "LAxisCtrl_typeMoveVelocity";   // Configuration of MC_MOVEVELOCITY function
      stop : "LAxisCtrl_typeStop";   // Configuration of MC_HALT function
      fastStop : "LAxisCtrl_typeFastStop";   // Configuration of MC_HALT function (alternative dynamics)
      torqueLimiting : "LAxisCtrl_typeTorqueLimiting";   // Configuration of MC_TORQUELIMITING function
      homing : "LAxisCtrl_typeHoming";   // Configuration of HOMING function
      posRelative : "LAxisCtrl_typePosRelative";   // Configuration of MC_MOVERELATIVE function
      posAbsolute : "LAxisCtrl_typePosAbsolute";   // Configuration of MC_MOVEABSOLUTE function
      posSuperimposed : "LAxisCtrl_typePosSuperimposed";   // Configuration of MC_MOVESUPERIMPOSED function
      gearInRelative : "LAxisCtrl_typeGearInRelative";   // Configuration of MC_GEARIN function
      gearInAbsolute : "LAxisCtrl_typeGearInAbsolute";   // Configuration of MC_GEARIN_POS function
      camIn : "LAxisCtrl_typeCamIn";   // Configuration of MC_CAMIN function
      gearOutCamOut : "LAxisCtrl_typeGearOutCamOut";   // Configuration of MC_GEAROUT / MC_CAMOUT function
      phasing : "LAxisCtrl_typePhasing";   // Configuration of MC_PHASING function
      offset : "LAxisCtrl_typeOffset";   // Configuration of MC_OFFSET function
   END_STRUCT;
END_TYPE

// ===== library: MasterCopy "LAxisCtrl_typeDiagnostics" =====

// folder: LAxisCtrl_Types

TYPE "LAxisCtrl_typeDiagnostics"
TITLE = LAxisCtrl_typeDiagnostics
// Support: tech.team.motioncontrol@siemens.com
   STRUCT
      status : Word := 16#0000;   // Status of FB when error occurred
      subfunctionStatus : Word := 16#0000;   // ErrorID of called subfunction
      basicMotionState : DInt := 0;   // Current basic motion state when error occurred
      superimposedMotionState : DInt := 0;   // Current superimposed motion state when error occurred
   END_STRUCT;
END_TYPE

// ===== library: MasterCopy "LAxisCtrl_AxisErrorWord" =====

// folder: LAxisCtrl_Blocks/AdditionalFunctions

FUNCTION_BLOCK "LAxisCtrl_AxisErrorWord"   // FB30615, SCL
TITLE = LAxisCtrl_AxisErrorWord
{ S7_Optimized_Access := 'TRUE' }
AUTHOR : tech.team.motioncontrol@siemens.com
FAMILY : AxisCtrl
VERSION : 1.1
// Support: tech.team.motioncontrol@siemens.com
   VAR_INPUT
      axis : DB_ANY;   // Axis specification
   END_VAR
   VAR_OUTPUT
      status : Word;   // Status of FB
      errorWord : DWord;   // ErrorWord of axis
      systemFault : Bool;   // TRUE: System fault (A system-internal error has occurred)
      configFault : Bool;   // TRUE: Configuration error (One or more configuration parameters are inconsistent or invalid)
      userFault : Bool;   // TRUE: User fault (Error in user program at a Motion Control instruction or its use)
      commandNotAccepted : Bool;   // TRUE: Job cannot be executed. A Motion Control instruction cannot be executed because the necessary conditions are not met
      driveFault : Bool;   // TRUE: Error in drive
      sensorFault : Bool;   // TRUE: Error in encoder system
      dynamicError : Bool;   // TRUE: Specified dynamic values are limited to permissible values
      communicationFault : Bool;   // TRUE: Communication error (Missing or faulty communication)
      swLimit : Bool;   // TRUE: Software limit switch reached or overtraveled
      hwLimit : Bool;   // TRUE: Hardware limit switch reached or overtraveled
      homingError : Bool;   // TRUE: Error during homing operation (The homing cannot be completed)
      followingErrorFault : Bool;   // TRUE: Following error limits exceeded
      positioningFault : Bool;   // TRUE: Positioning error
      peripheralError : Bool;   // TRUE: Error accessing a logical address
      synchronousError : Bool;   // TRUE: Error during synchronous operation (The leading axis specified for the Motion Control instruction was not configured as a possible leading axis)
      adaptionError : Bool;   // TRUE: Error in automatic data transfer
   END_VAR
   VAR_TEMP
      tempErrorWord : DWord;   // Temporary errorWord
   END_VAR
   VAR CONSTANT
      ERROR_INVALID_TECHNOLOGY_OBJECT : Word := 16#8002;   // Illegal specification of the technology object. Check the specification of the technology object for the "Axis", "Master" or "Cam" parameter.
      FINISHED : Word;   // FB Finished
   END_VAR
BEGIN
   REGION HEADER
     //================================================================================
     // SIEMENS AG
     // (c)Copyright 2020 All Rights Reserved
     //--------------------------------------------------------------------------------
     // Library: LAxisCtrl 
     // Tested with: S7-1515-2 PN
     // Engineering: TIA Portal V16
     // Restrictions: -
     // Requirements: S7-1500 FW 2.8.1
     // Functionality: The FB is splitting the error word of an axis (DB_Any) into bits.
     // Support: tech.team.motioncontrol@siemens.com
     // Note: Parameter comments are only available in language 'English (United States)'
     //--------------------------------------------------------------------------------
     // Change log table:
     // Version  Date        Expert in charge  Changes applied
     // 01.01.00 12.03.2020  RS                First released version
     //================================================================================
   END_REGION

   CASE TypeOfDB(#axis) OF
     TO_ExternalEncoder:
       #tempErrorWord := "LAxisCtrl_UnpubErrorWordExtEncoder"(#axis);
       #status := #FINISHED;

     TO_SpeedAxis:
       #tempErrorWord := "LAxisCtrl_UnpubErrorWordSpeedAxis"(#axis);
       #status := #FINISHED;

     TO_PositioningAxis:
       #tempErrorWord := "LAxisCtrl_UnpubErrorWordPosAxis"(#axis);
       #status := #FINISHED;

     TO_SynchronousAxis:
       #tempErrorWord := "LAxisCtrl_UnpubErrorWordSyncAxis"(#axis);
       #status := #FINISHED;

     ELSE
       #tempErrorWord := 16#0000_0000;
       #status := #ERROR_INVALID_TECHNOLOGY_OBJECT;
       ENO := FALSE;
   END_CASE;

   #errorWord := #tempErrorWord;
   //----------------------------------------------------------------------------------------------
   // Write outputs
   //----------------------------------------------------------------------------------------------
   #systemFault := #tempErrorWord.%X0;
   #configFault := #tempErrorWord.%X1;
   #userFault := #tempErrorWord.%X2;
   #commandNotAccepted := #tempErrorWord.%X3;
   #driveFault := #tempErrorWord.%X4;
   #sensorFault := #tempErrorWord.%X5;
   #dynamicError := #tempErrorWord.%X6;
   #communicationFault := #tempErrorWord.%X7;
   #swLimit := #tempErrorWord.%X8;
   #hwLimit := #tempErrorWord.%X9;
   #homingError := #tempErrorWord.%X10;
   #followingErrorFault := #tempErrorWord.%X11;
   #positioningFault := #tempErrorWord.%X12;
   #peripheralError := #tempErrorWord.%X13;
   #synchronousError := #tempErrorWord.%X14;
   #adaptionError := #tempErrorWord.%X15;
END_FUNCTION_BLOCK

// ===== library: MasterCopy "LAxisCtrl_AxisStatusWord" =====

// folder: LAxisCtrl_Blocks/AdditionalFunctions

FUNCTION_BLOCK "LAxisCtrl_AxisStatusWord"   // FB30613, SCL
TITLE = LAxisCtrl_AxisStatusWord
{ S7_Optimized_Access := 'TRUE' }
AUTHOR : tech.team.motioncontrol@siemens.com
FAMILY : AxisCtrl
VERSION : 1.2
// Support: tech.team.motioncontrol@siemens.com
   VAR_INPUT
      axis : DB_ANY;   // Axis specification
   END_VAR
   VAR_OUTPUT
      status : Word;   // Status of FB
      statusWord : DWord;   // StatusWord of axis
      statusWord2 : DWord;   // StatusWord2 of axis
      enable : Bool;   // TRUE: Technology object is enabled
      error : Bool;   // TRUE: An error is present
      restartActive : Bool;   // TRUE: A restart is active. The technology object is being reinitialized
      onlineStartValuesChanged : Bool;   // TRUE: The restart tags have been changed. For the changes to be applied, the technology object must be reinitialized
      controlPanelActive : Bool;   // TRUE: Axis control panel is active
      homingDone : Bool;   // TRUE: The technology object is homed
      done : Bool;   // TRUE: No motion job is in progress and the axis control panel is deactivated
      standstill : Bool;   // TRUE: The axis is at a standstill
      positioningCommand : Bool;   // TRUE: A positioning job is running ("MC_MoveRelative", "MC_MoveAbsolute")
      jogCommand : Bool;   // TRUE: A "MC_MoveJog" job is running
      velocityCommand : Bool;   // TRUE: A "MC_MoveVelocity" job is running
      homingCommand : Bool;   // TRUE: A "MC_Home" job is being processed
      constantVelocity : Bool;   // TRUE: The setpoint velocity is reached. The axis is traversing at this constant velocity or is at a standstill
      accelerating : Bool;   // TRUE: An acceleration process is active
      decelerating : Bool;   // TRUE: A deceleration process is active
      swLimitMinActive : Bool;   // TRUE: A negative software limit switch was reached or exceeded
      swLimitMaxActive : Bool;   // TRUE: A positive software limit switch was reached or exceeded
      hwLimitMinActive : Bool;   // TRUE: A negative hardware limit switch was reached or exceeded
      hwLimitMaxActive : Bool;   // TRUE: A positive hardware limit switch was reached or exceeded
      synchronizing : Bool;   // TRUE: The axis synchronizes to a leading value
      synchronous : Bool;   // TRUE: The axis moves synchronously to a leading value
      superimposedMotionCommand : Bool;   // TRUE: A superimposed motion is active
      phasingCommand : Bool;   // TRUE: A Motion Control instruction for leading value shift is active
      axisSimulation : Bool;   // TRUE: The technology object is in simulation
      torqueLimitingCommand : Bool;   // TRUE: A "MC_TorqueLimiting" job is running
      inLimitation : Bool;   // TRUE: The drive is operating at the torque limit
      nonPositionControlled : Bool;   // TRUE: The axis is in non position-controlled mode
      kinematicsMotionCommand : Bool;   // TRUE: The axis is used for a kinematics job
      inClamping : Bool;   // TRUE: The axis is clamped at a fixed stop
      motionInCommand : Bool;   // TRUE: A "MC_MotionIn" job is active
      stopCommand : Bool;   // TRUE: A "MC_Stop" job is running. The technology object is locked
      desynchronizingCommand : Bool;   // TRUE: A "MC_GearOut" job or "MC_CamOut" job is active. The following axis is desynchronized
      passingBacklash : Bool;   // TRUE: The backlash is traversed. <TO>.ActualPosition does not hereby change
      phasingCommandWaiting : Bool;   // TRUE: A "MC_PhasingAbsolute" or "MC_PhasingRelative" job for leading value shift is waiting
      offsetCommand : Bool;   // TRUE: A "MC_OffsetAbsolute" or "MC_OffsetRelative" job for following value offset is active
      offsetCommandWaiting : Bool;   // TRUE: A "MC_OffsetAbsolute" or "MC_OffsetRelative" job for following value offset is waiting
   END_VAR
   VAR_TEMP
      tempStatusWord : DWord;   // Temporary statusWord
      tempStatusWord2 : DWord;   // Temporary statusWord2
   END_VAR
   VAR CONSTANT
      ERROR_INVALID_TECHNOLOGY_OBJECT : Word := 16#8002;   // Illegal specification of the technology object. Check the specification of the technology object for the "Axis", "Master" or "Cam" parameter.
      FINISHED : Word;   // FB Finished
   END_VAR
BEGIN
   REGION HEADER
     //================================================================================
     // SIEMENS AG
     // (c)Copyright 2021 All Rights Reserved
     //--------------------------------------------------------------------------------
     // Library: LAxisCtrl
     // Tested with: S7-1515-2 PN
     // Engineering: TIA Portal V17
     // Restrictions: -
     // Requirements: S7-1500 FW 2.9
     //               LAnyAxis V1.1        
     // Functionality: The FB is splitting the status word of an axis (DB_Any) into bits.
     // Support: tech.team.motioncontrol@siemens.com
     // Note: Parameter comments are only available in language 'English (United States)'
     //--------------------------------------------------------------------------------
     // Change log table:
     // Version  Date        Expert in charge  Changes applied
     // 01.01.00 12.03.2020  RS                First released version
     // 01.02.00 09.03.2021  RS                Update Motion Control V6.0
     //================================================================================
   END_REGION

   CASE TypeOfDB(#axis) OF
     TO_ExternalEncoder:
       #tempStatusWord := "LAnyAxis_UnpubStatusWordExtEncoder"(#axis);
       #tempStatusWord2 := 16#0000_0000;
       #status := #FINISHED;

     TO_SpeedAxis:
       #tempStatusWord := "LAnyAxis_UnpubStatusWordSpeedAxis"(#axis);
       #tempStatusWord2 := "LAnyAxis_UnpubStatusWord2SpeedAxis"(#axis);
       #status := #FINISHED;

     TO_PositioningAxis:
       #tempStatusWord := "LAnyAxis_UnpubStatusWordPosAxis"(#axis);
       #tempStatusWord2 := "LAnyAxis_UnpubStatusWord2PosAxis"(#axis);
       #status := #FINISHED;

     TO_SynchronousAxis:
       #tempStatusWord := "LAnyAxis_UnpubStatusWordSyncAxis"(#axis);
       #tempStatusWord2 := "LAnyAxis_UnpubStatusWord2SyncAxis"(#axis);
       #status := #FINISHED;

     ELSE
       #tempStatusWord := 16#0000_0000;
       #tempStatusWord2 := 16#0000_0000;
       #status := #ERROR_INVALID_TECHNOLOGY_OBJECT;
   END_CASE;

   #statusWord := #tempStatusWord;
   #statusWord2 := #tempStatusWord2;
   //----------------------------------------------------------------------------------------------
   // Write outputs
   //----------------------------------------------------------------------------------------------
   #enable                    := #tempStatusWord.%X0;
   #error                     := #tempStatusWord.%X1;
   #restartActive             := #tempStatusWord.%X2;
   #onlineStartValuesChanged  := #tempStatusWord.%X3;
   #controlPanelActive        := #tempStatusWord.%X4;
   #homingDone                := #tempStatusWord.%X5;
   #done                      := #tempStatusWord.%X6;
   #standstill                := #tempStatusWord.%X7;
   #positioningCommand        := #tempStatusWord.%X8;
   #jogCommand                := #tempStatusWord.%X9;
   #velocityCommand           := #tempStatusWord.%X10;
   #homingCommand             := #tempStatusWord.%X11;
   #constantVelocity          := #tempStatusWord.%X12;
   #accelerating              := #tempStatusWord.%X13;
   #decelerating              := #tempStatusWord.%X14;
   #swLimitMinActive          := #tempStatusWord.%X15;
   #swLimitMaxActive          := #tempStatusWord.%X16;
   #hwLimitMinActive          := #tempStatusWord.%X17;
   #hwLimitMaxActive          := #tempStatusWord.%X18;
   #synchronizing             := #tempStatusWord.%X21;
   #synchronous               := #tempStatusWord.%X22;
   #superimposedMotionCommand := #tempStatusWord.%X23;
   #phasingCommand            := #tempStatusWord.%X24;
   #axisSimulation            := #tempStatusWord.%X25;
   #torqueLimitingCommand     := #tempStatusWord.%X26;
   #inLimitation              := #tempStatusWord.%X27;
   #nonPositionControlled     := #tempStatusWord.%X28;
   #kinematicsMotionCommand   := #tempStatusWord.%X29; // V15
   #inClamping                := #tempStatusWord.%X30;
   #motionInCommand           := #tempStatusWord.%X31; // V15

   #stopCommand               := #tempStatusWord2.%X0; // V16

   #desynchronizingCommand    := #tempStatusWord2.%X1; // V17
   #passingBacklash           := #tempStatusWord2.%X2; // V17
   #phasingCommandWaiting     := #tempStatusWord2.%X3; // V17
   #offsetCommand             := #tempStatusWord2.%X4; // V17
   #offsetCommandWaiting      := #tempStatusWord2.%X5; // V17
END_FUNCTION_BLOCK

// ===== library: MasterCopy "LAxisCtrl_AxisWarningWord" =====

// folder: LAxisCtrl_Blocks/AdditionalFunctions

FUNCTION_BLOCK "LAxisCtrl_AxisWarningWord"   // FB30614, SCL
TITLE = LAxisCtrl_AxisWarningWord
{ S7_Optimized_Access := 'TRUE' }
AUTHOR : tech.team.motioncontrol@siemens.com
FAMILY : AxisCtrl
VERSION : 1.1
// Support: tech.team.motioncontrol@siemens.com
   VAR_INPUT
      axis : DB_ANY;   // Axis specification
   END_VAR
   VAR_OUTPUT
      status : Word;   // Status of FB
      warningWord : DWord;   // WarningWord of axis
      systemWarning : Bool;   // TRUE: A system-internal error has occurred
      configWarning : Bool;   // TRUE: Configuration error (One or several configuration parameters are adjusted internally)
      userWarning : Bool;   // TRUE: Error in user program at a Motion Control instruction or its use
      commandNotAccepted : Bool;   // TRUE: Job cannot be executed. A Motion Control instruction cannot be executed because the necessary conditions are not met
      driveWarning : Bool;   // TRUE: Warning in drive
      sensorWarning : Bool;   // TRUE: Error in encoder system
      dynamicError : Bool;   // TRUE: Specified dynamic values are limited to permissible values
      communicationWarning : Bool;   // TRUE: Communication error (Missing or faulty communication)
      swLimitMin : Bool;   // TRUE: The negative software limit switch has been approached
      swLimitMax : Bool;   // TRUE: The positive software limit switch has been approached
      homingWarning : Bool;   // TRUE: Error during homing operation (The homing cannot be completed)
      followingErrorWarning : Bool;   // TRUE: Warning limit of following error monitoring reached/exceeded
      positioningWarning : Bool;   // TRUE: Positioning error
      peripheralWarning : Bool;   // TRUE: Error accessing a logical address
      synchronousWarning : Bool;   // TRUE: Error during synchronous operation (The leading axis specified for the Motion Control instruction was not configured as a possible leading axis)
      adaptionWarning : Bool;   // TRUE: Error in automatic data transfer
   END_VAR
   VAR_TEMP
      tempWarningWord : DWord;   // Temporary warningWord
   END_VAR
   VAR CONSTANT
      ERROR_INVALID_TECHNOLOGY_OBJECT : Word := 16#8002;   // Illegal specification of the technology object. Check the specification of the technology object for the "Axis", "Master" or "Cam" parameter.
      FINISHED : Word;   // FB Finished
   END_VAR
BEGIN
   REGION HEADER
     //================================================================================
     // SIEMENS AG
     // (c)Copyright 2020 All Rights Reserved
     //--------------------------------------------------------------------------------
     // Library: LAxisCtrl 
     // Tested with: S7-1515-2 PN
     // Engineering: TIA Portal V16
     // Restrictions: -
     // Requirements: S7-1500 FW 2.8.1
     // Functionality: The FB is splitting the warning word of an axis (DB_Any) into bits.
     // Support: tech.team.motioncontrol@siemens.com
     // Note: Parameter comments are only available in language 'English (United States)'
     //--------------------------------------------------------------------------------
     // Change log table:
     // Version  Date        Expert in charge  Changes applied
     // 01.01.00 12.03.2020  RS                First released version
     //================================================================================
   END_REGION

   CASE TypeOfDB(#axis) OF
     TO_ExternalEncoder:
       #tempWarningWord := "LAxisCtrl_UnpubWarningWordExtEncoder"(#axis);
       #status := #FINISHED;

     TO_SpeedAxis:
       #tempWarningWord := "LAxisCtrl_UnpubWarningWordSpeedAxis"(#axis);
       #status := #FINISHED;

     TO_PositioningAxis:
       #tempWarningWord := "LAxisCtrl_UnpubWarningWordPosAxis"(#axis);
       #status := #FINISHED;

     TO_SynchronousAxis:
       #tempWarningWord := "LAxisCtrl_UnpubWarningWordSyncAxis"(#axis);
       #status := #FINISHED;

     ELSE
       #tempWarningWord := 16#0000_0000;
       #status := #ERROR_INVALID_TECHNOLOGY_OBJECT;
       ENO := FALSE;
   END_CASE;

   #warningWord := #tempWarningWord;
   //----------------------------------------------------------------------------------------------
   // Write outputs
   //----------------------------------------------------------------------------------------------
   #systemWarning := #tempWarningWord.%X0;
   #configWarning := #tempWarningWord.%X1;
   #userWarning := #tempWarningWord.%X2;
   #commandNotAccepted := #tempWarningWord.%X3;
   #driveWarning := #tempWarningWord.%X4;
   #sensorWarning := #tempWarningWord.%X5;
   #dynamicError := #tempWarningWord.%X6;
   #communicationWarning := #tempWarningWord.%X7;
   #swLimitMin := #tempWarningWord.%X8;
   #swLimitMax := #tempWarningWord.%X9;
   #homingWarning := #tempWarningWord.%X10;
   #followingErrorWarning := #tempWarningWord.%X11;
   #positioningWarning := #tempWarningWord.%X12;
   #peripheralWarning := #tempWarningWord.%X13;
   #synchronousWarning := #tempWarningWord.%X14;
   #adaptionWarning := #tempWarningWord.%X15;
END_FUNCTION_BLOCK

// ===== library: MasterCopy "LAxisCtrl_UnpubErrorWordExtEncoder" =====

// folder: LAxisCtrl_Blocks/AdditionalFunctions/InternalSubBlocks/ErrorWord

FUNCTION "LAxisCtrl_UnpubErrorWordExtEncoder" : DWord   // FC30600, SCL
TITLE = LAxisCtrl_UnpubErrorWordExtEncoder
{ S7_Optimized_Access := 'TRUE' }
AUTHOR : tech.team.motioncontrol@siemens.com
FAMILY : AxisCtrl
VERSION : 1.1
// Support: tech.team.motioncontrol@siemens.com
   VAR_INPUT
      axis : TO_ExternalEncoder;   // Axis specification
   END_VAR
   // Ret_Val : axis.ErrorWord
BEGIN
   // Read axis parameter
   #LAxisCtrl_UnpubErrorWordExtEncoder := #axis.ErrorWord;
END_FUNCTION

// ===== library: MasterCopy "LAxisCtrl_UnpubErrorWordPosAxis" =====

// folder: LAxisCtrl_Blocks/AdditionalFunctions/InternalSubBlocks/ErrorWord

FUNCTION "LAxisCtrl_UnpubErrorWordPosAxis" : DWord   // FC30601, SCL
TITLE = LAxisCtrl_UnpubErrorWordPosAxis
{ S7_Optimized_Access := 'TRUE' }
AUTHOR : tech.team.motioncontrol@siemens.com
FAMILY : AxisCtrl
VERSION : 1.1
// Support: tech.team.motioncontrol@siemens.com
   VAR_INPUT
      axis : TO_PositioningAxis;   // Axis specification
   END_VAR
   // Ret_Val : axis.ErrorWord
BEGIN
   // Read axis parameter
   #LAxisCtrl_UnpubErrorWordPosAxis := #axis.ErrorWord;
END_FUNCTION

// ===== library: MasterCopy "LAxisCtrl_UnpubErrorWordSpeedAxis" =====

// folder: LAxisCtrl_Blocks/AdditionalFunctions/InternalSubBlocks/ErrorWord

FUNCTION "LAxisCtrl_UnpubErrorWordSpeedAxis" : DWord   // FC30602, SCL
TITLE = LAxisCtrl_UnpubErrorWordSpeedAxis
{ S7_Optimized_Access := 'TRUE' }
AUTHOR : tech.team.motioncontrol@siemens.com
FAMILY : AxisCtrl
VERSION : 1.1
// Support: tech.team.motioncontrol@siemens.com
   VAR_INPUT
      axis : TO_SpeedAxis;   // Axis specification
   END_VAR
   // Ret_Val : axis.ErrorWord
BEGIN
   // Read axis parameter
   #LAxisCtrl_UnpubErrorWordSpeedAxis := #axis.ErrorWord;
END_FUNCTION

// ===== library: MasterCopy "LAxisCtrl_UnpubErrorWordSyncAxis" =====

// folder: LAxisCtrl_Blocks/AdditionalFunctions/InternalSubBlocks/ErrorWord

FUNCTION "LAxisCtrl_UnpubErrorWordSyncAxis" : DWord   // FC30603, SCL
TITLE = LAxisCtrl_UnpubErrorWordSyncAxis
{ S7_Optimized_Access := 'TRUE' }
AUTHOR : tech.team.motioncontrol@siemens.com
FAMILY : AxisCtrl
VERSION : 1.1
// Support: tech.team.motioncontrol@siemens.com
   VAR_INPUT
      axis : TO_SynchronousAxis;   // Axis specification
   END_VAR
   // Ret_Val : axis.ErrorWord
BEGIN
   // Read axis parameter
   #LAxisCtrl_UnpubErrorWordSyncAxis := #axis.ErrorWord;
END_FUNCTION

// ===== library: MasterCopy "LAxisCtrl_UnpubWarningWordExtEncoder" =====

// folder: LAxisCtrl_Blocks/AdditionalFunctions/InternalSubBlocks/WarningWord

FUNCTION "LAxisCtrl_UnpubWarningWordExtEncoder" : DWord   // FC30608, SCL
TITLE = LAxisCtrl_UnpubWarningWordExtEncoder
{ S7_Optimized_Access := 'TRUE' }
AUTHOR : tech.team.motioncontrol@siemens.com
FAMILY : AxisCtrl
VERSION : 1.1
// Support: tech.team.motioncontrol@siemens.com
   VAR_INPUT
      axis : TO_ExternalEncoder;   // Axis specification
   END_VAR
   // Ret_Val : axis.WarningWord
BEGIN
   // Read axis parameter
   #LAxisCtrl_UnpubWarningWordExtEncoder := #axis.WarningWord;
END_FUNCTION

// ===== library: MasterCopy "LAxisCtrl_UnpubWarningWordPosAxis" =====

// folder: LAxisCtrl_Blocks/AdditionalFunctions/InternalSubBlocks/WarningWord

FUNCTION "LAxisCtrl_UnpubWarningWordPosAxis" : DWord   // FC30609, SCL
TITLE = LAxisCtrl_UnpubWarningWordPosAxis
{ S7_Optimized_Access := 'TRUE' }
AUTHOR : tech.team.motioncontrol@siemens.com
FAMILY : AxisCtrl
VERSION : 1.1
// Support: tech.team.motioncontrol@siemens.com
   VAR_INPUT
      axis : TO_PositioningAxis;   // Axis specification
   END_VAR
   // Ret_Val : axis.WarningWord
BEGIN
   // Read axis parameter
   #LAxisCtrl_UnpubWarningWordPosAxis := #axis.WarningWord;
END_FUNCTION

// ===== library: MasterCopy "LAxisCtrl_UnpubWarningWordSpeedAxis" =====

// folder: LAxisCtrl_Blocks/AdditionalFunctions/InternalSubBlocks/WarningWord

FUNCTION "LAxisCtrl_UnpubWarningWordSpeedAxis" : DWord   // FC30610, SCL
TITLE = LAxisCtrl_UnpubWarningWordSpeedAxis
{ S7_Optimized_Access := 'TRUE' }
AUTHOR : tech.team.motioncontrol@siemens.com
FAMILY : AxisCtrl
VERSION : 1.1
// Support: tech.team.motioncontrol@siemens.com
   VAR_INPUT
      axis : TO_SpeedAxis;   // Axis specification
   END_VAR
   // Ret_Val : axis.WarningWord
BEGIN
   // Read axis parameter
   #LAxisCtrl_UnpubWarningWordSpeedAxis := #axis.WarningWord;
END_FUNCTION

// ===== library: MasterCopy "LAxisCtrl_UnpubWarningWordSyncAxis" =====

// folder: LAxisCtrl_Blocks/AdditionalFunctions/InternalSubBlocks/WarningWord

FUNCTION "LAxisCtrl_UnpubWarningWordSyncAxis" : DWord   // FC30611, SCL
TITLE = LAxisCtrl_UnpubWarningWordSyncAxis
{ S7_Optimized_Access := 'TRUE' }
AUTHOR : tech.team.motioncontrol@siemens.com
FAMILY : AxisCtrl
VERSION : 1.1
// Support: tech.team.motioncontrol@siemens.com
   VAR_INPUT
      axis : TO_SynchronousAxis;   // Axis specification
   END_VAR
   // Ret_Val : axis.WarningWord
BEGIN
   // Read axis parameter
   #LAxisCtrl_UnpubWarningWordSyncAxis := #axis.WarningWord;
END_FUNCTION

// ===== library: MasterCopy "LAxisCtrl_UnpubAxisDynamicDefaultAcc" =====

// folder: LAxisCtrl_Blocks/InternalSubBlocks

FUNCTION "LAxisCtrl_UnpubAxisDynamicDefaultAcc" : LReal   // FC30613, SCL
TITLE = LAxisCtrl_UnpubAxisDynamicDefaultAcc
{ S7_Optimized_Access := 'TRUE' }
AUTHOR : tech.team.motioncontrol@siemens.com
FAMILY : AxisCtrl
VERSION : 1.1
// Support: tech.team.motioncontrol@siemens.com
   VAR_INPUT
      axis : DB_ANY;   // Axis specification
   END_VAR
   // Ret_Val : axis.DynamicDefaults.Acceleration
BEGIN
   // Read axis parameter
   CASE TypeOfDB(#axis) OF
     TO_PositioningAxis:
       #LAxisCtrl_UnpubAxisDynamicDefaultAcc := "LAxisCtrl_UnpubDynamicDefaultAccPosAxis"(#axis);

     TO_SynchronousAxis:
       #LAxisCtrl_UnpubAxisDynamicDefaultAcc := "LAxisCtrl_UnpubDynamicDefaultAccSyncAxis"(#axis);

     ELSE
       #LAxisCtrl_UnpubAxisDynamicDefaultAcc := -1.0;
   END_CASE;
END_FUNCTION

// ===== library: MasterCopy "LAxisCtrl_UnpubAxisDynamicDefaultDec" =====

// folder: LAxisCtrl_Blocks/InternalSubBlocks

FUNCTION "LAxisCtrl_UnpubAxisDynamicDefaultDec" : LReal   // FC30621, SCL
TITLE = LAxisCtrl_UnpubAxisDynamicDefaultDec
{ S7_Optimized_Access := 'TRUE' }
AUTHOR : tech.team.motioncontrol@siemens.com
FAMILY : AxisCtrl
VERSION : 1.1
// Support: tech.team.motioncontrol@siemens.com
   VAR_INPUT
      axis : DB_ANY;   // Axis specification
   END_VAR
   // Ret_Val : axis.DynamicDefaults.Deceleration
BEGIN
   // Read axis parameter
   CASE TypeOfDB(#axis) OF
     TO_PositioningAxis:
       #LAxisCtrl_UnpubAxisDynamicDefaultDec := "LAxisCtrl_UnpubDynamicDefaultDecPosAxis"(#axis);

     TO_SynchronousAxis:
       #LAxisCtrl_UnpubAxisDynamicDefaultDec := "LAxisCtrl_UnpubDynamicDefaultDecSyncAxis"(#axis);

     ELSE
       #LAxisCtrl_UnpubAxisDynamicDefaultDec := -1.0;
   END_CASE;
END_FUNCTION

// ===== library: MasterCopy "LAxisCtrl_UnpubAxisDynamicDefaultJerk" =====

// folder: LAxisCtrl_Blocks/InternalSubBlocks

FUNCTION "LAxisCtrl_UnpubAxisDynamicDefaultJerk" : LReal   // FC30646, SCL
TITLE = LAxisCtrl_UnpubAxisDynamicDefaultJerk
{ S7_Optimized_Access := 'TRUE' }
AUTHOR : tech.team.motioncontrol@siemens.com
FAMILY : AxisCtrl
VERSION : 1.1
// Support: tech.team.motioncontrol@siemens.com
   VAR_INPUT
      axis : DB_ANY;   // Axis specification
   END_VAR
   // Ret_Val : axis.DynamicDefaults.Jerk
BEGIN
   // Read axis parameter
   CASE TypeOfDB(#axis) OF
     TO_PositioningAxis:
       #LAxisCtrl_UnpubAxisDynamicDefaultJerk := "LAxisCtrl_UnpubDynamicDefaultJerkPosAxis"(#axis);

     TO_SynchronousAxis:
       #LAxisCtrl_UnpubAxisDynamicDefaultJerk := "LAxisCtrl_UnpubDynamicDefaultJerkSyncAxis"(#axis);

     ELSE
       #LAxisCtrl_UnpubAxisDynamicDefaultJerk := 0.0; // No Jerk
   END_CASE;
END_FUNCTION

// ===== library: MasterCopy "LAxisCtrl_UnpubAxisEmergencyDec" =====

// folder: LAxisCtrl_Blocks/InternalSubBlocks

FUNCTION "LAxisCtrl_UnpubAxisEmergencyDec" : LReal   // FC30614, SCL
TITLE = LAxisCtrl_UnpubAxisEmergencyDec
{ S7_Optimized_Access := 'TRUE' }
AUTHOR : tech.team.motioncontrol@siemens.com
FAMILY : AxisCtrl
VERSION : 1.1
// Support: tech.team.motioncontrol@siemens.com
   VAR_INPUT
      axis : DB_ANY;   // Axis specification
   END_VAR
   // Ret_Val : axis.DynamicDefaults.EmergencyDeceleration
BEGIN
   // Read axis parameter
   CASE TypeOfDB(#axis) OF
     TO_SpeedAxis:
       #LAxisCtrl_UnpubAxisEmergencyDec := "LAxisCtrl_UnpubEmergencyDecSpeedAxis"(#axis);

     TO_PositioningAxis:
       #LAxisCtrl_UnpubAxisEmergencyDec := "LAxisCtrl_UnpubEmergencyDecPosAxis"(#axis);

     TO_SynchronousAxis:
       #LAxisCtrl_UnpubAxisEmergencyDec := "LAxisCtrl_UnpubEmergencyDecSyncAxis"(#axis);

     ELSE
       #LAxisCtrl_UnpubAxisEmergencyDec := -1.0; 
   END_CASE;
END_FUNCTION

// ===== library: MasterCopy "LAxisCtrl_UnpubAxisHomingDirection" =====

// folder: LAxisCtrl_Blocks/InternalSubBlocks

FUNCTION "LAxisCtrl_UnpubAxisHomingDirection" : DInt   // FC30612, SCL
TITLE = LAxisCtrl_UnpubAxisHomingDirection
{ S7_Optimized_Access := 'TRUE' }
AUTHOR : tech.team.motioncontrol@siemens.com
FAMILY : AxisCtrl
VERSION : 1.1
// Support: tech.team.motioncontrol@siemens.com
   VAR_INPUT
      axis : DB_ANY;   // Axis specification
      index : Int;   // Index of sensor
   END_VAR
   // Ret_Val : axis.Sensor[index].ActiveHoming.Direction
BEGIN
   // Read axis parameter
   CASE TypeOfDB(#axis) OF
     TO_PositioningAxis:
       #LAxisCtrl_UnpubAxisHomingDirection := "LAxisCtrl_UnpubHomingDirectionPosAxis"(axis := #axis, index := #index);

     TO_SynchronousAxis:
       #LAxisCtrl_UnpubAxisHomingDirection := "LAxisCtrl_UnpubHomingDirectionSyncAxis"(axis := #axis, index := #index);

     ELSE
       #LAxisCtrl_UnpubAxisHomingDirection := 0; // Positive direction
   END_CASE;
END_FUNCTION

// ===== library: MasterCopy "LAxisCtrl_UnpubAxisModuloEnabled" =====

// folder: LAxisCtrl_Blocks/InternalSubBlocks

FUNCTION "LAxisCtrl_UnpubAxisModuloEnabled" : Bool   // FC30627, SCL
TITLE = LAxisCtrl_UnpubAxisModuloEnabled
{ S7_Optimized_Access := 'TRUE' }
AUTHOR : tech.team.motioncontrol@siemens.com
FAMILY : AxisCtrl
VERSION : 1.1
// Support: tech.team.motioncontrol@siemens.com
   VAR_INPUT
      axis : DB_ANY;   // Axis specification
   END_VAR
   // Ret_Val : axis.Modulo.Enable
BEGIN
   // Read axis parameter
   CASE TypeOfDB(#axis) OF
     TO_PositioningAxis:
       #LAxisCtrl_UnpubAxisModuloEnabled := "LAnyAxis_UnpubModuloEnablePosAxis"(#axis);

     TO_SynchronousAxis:
       #LAxisCtrl_UnpubAxisModuloEnabled := "LAnyAxis_UnpubModuloEnableSyncAxis"(#axis);

     TO_ExternalEncoder:
       #LAxisCtrl_UnpubAxisModuloEnabled := "LAnyAxis_UnpubModuloEnableExtEncoder"(#axis);

     ELSE
       #LAxisCtrl_UnpubAxisModuloEnabled := FALSE;
   END_CASE;
END_FUNCTION

// ===== library: MasterCopy "LAxisCtrl_UnpubAxisOperativeSensor" =====

// folder: LAxisCtrl_Blocks/InternalSubBlocks

FUNCTION "LAxisCtrl_UnpubAxisOperativeSensor" : UDInt   // FC30644, SCL
TITLE = LAxisCtrl_UnpubAxisOperativeSensor
{ S7_Optimized_Access := 'TRUE' }
AUTHOR : tech.team.motioncontrol@siemens.com
FAMILY : AxisCtrl
VERSION : 1.1
// Support: tech.team.motioncontrol@siemens.com
   VAR_INPUT
      axis : DB_ANY;   // Axis specification
   END_VAR
   // Ret_Val : axis.OperativeSensor
BEGIN
   // Read axis parameter
   CASE TypeOfDB(#axis) OF
     TO_PositioningAxis:
       #LAxisCtrl_UnpubAxisOperativeSensor := "LAxisCtrl_UnpubOperativeSensorPosAxis"(axis := #axis);

     TO_SynchronousAxis:
       #LAxisCtrl_UnpubAxisOperativeSensor := "LAxisCtrl_UnpubOperativeSensorSyncAxis"(axis := #axis);

     ELSE
       #LAxisCtrl_UnpubAxisOperativeSensor := 1;
   END_CASE;
END_FUNCTION

// ===== library: MasterCopy "LAxisCtrl_UnpubAxisPosition" =====

// folder: LAxisCtrl_Blocks/InternalSubBlocks

FUNCTION "LAxisCtrl_UnpubAxisPosition" : LReal   // FC30615, SCL
TITLE = LAxisCtrl_UnpubAxisPosition
{ S7_Optimized_Access := 'TRUE' }
AUTHOR : tech.team.motioncontrol@siemens.com
FAMILY : AxisCtrl
VERSION : 1.1
// Support: tech.team.motioncontrol@siemens.com
   VAR_INPUT
      axis : DB_ANY;   // Axis specification
   END_VAR
   // Ret_Val : axis.Position
BEGIN
   // Read axis parameter
   CASE TypeOfDB(#axis) OF

     TO_PositioningAxis:
       #LAxisCtrl_UnpubAxisPosition := "LAnyAxis_UnpubPositionPosAxis"(#axis);

     TO_SynchronousAxis:
       #LAxisCtrl_UnpubAxisPosition := "LAnyAxis_UnpubPositionSyncAxis"(#axis);

     ELSE
       #LAxisCtrl_UnpubAxisPosition := 0.0;
   END_CASE;
END_FUNCTION

// ===== library: MasterCopy "LAxisCtrl_UnpubAxisPositioningDistance" =====

// folder: LAxisCtrl_Blocks/InternalSubBlocks

FUNCTION "LAxisCtrl_UnpubAxisPositioningDistance" : LReal   // FC30616, SCL
TITLE = LAxisCtrl_UnpubAxisPositioningDistance
{ S7_Optimized_Access := 'TRUE' }
AUTHOR : tech.team.motioncontrol@siemens.com
FAMILY : AxisCtrl
VERSION : 1.1
// Support: tech.team.motioncontrol@siemens.com
   VAR_INPUT
      axis : DB_ANY;   // Axis specification
   END_VAR
   // Ret_Val : axis.StatusPositioning.Distance
BEGIN
   // Read axis parameter
   CASE TypeOfDB(#axis) OF
     TO_PositioningAxis:
       #LAxisCtrl_UnpubAxisPositioningDistance := "LAxisCtrl_UnpubPositioningDistancePosAxis"(#axis);

     TO_SynchronousAxis:
       #LAxisCtrl_UnpubAxisPositioningDistance := "LAxisCtrl_UnpubPositioningDistanceSyncAxis"(#axis);

     ELSE
       #LAxisCtrl_UnpubAxisPositioningDistance := 0.0;
   END_CASE;
END_FUNCTION

// ===== library: MasterCopy "LAxisCtrl_UnpubAxisPositionTolerance" =====

// folder: LAxisCtrl_Blocks/InternalSubBlocks

FUNCTION "LAxisCtrl_UnpubAxisPositionTolerance" : LReal   // FC30617, SCL
TITLE = LAxisCtrl_UnpubAxisPositionTolerance
{ S7_Optimized_Access := 'TRUE' }
AUTHOR : tech.team.motioncontrol@siemens.com
FAMILY : AxisCtrl
VERSION : 1.1
// Support: tech.team.motioncontrol@siemens.com
   VAR_INPUT
      axis : DB_ANY;   // Axis specification
   END_VAR
   // Ret_Val : axis.Clamping.PositionTolerance
BEGIN
   // Read axis parameter
   CASE TypeOfDB(#axis) OF
     TO_PositioningAxis:
       #LAxisCtrl_UnpubAxisPositionTolerance := "LAxisCtrl_UnpubPositionTolerancePosAxis"(#axis);

     TO_SynchronousAxis:
       #LAxisCtrl_UnpubAxisPositionTolerance := "LAxisCtrl_UnpubPositionToleranceSyncAxis"(#axis);

     ELSE
       #LAxisCtrl_UnpubAxisPositionTolerance := 0.0;
   END_CASE;
END_FUNCTION

// ===== library: MasterCopy "LAxisCtrl_UnpubAxisReferencingVelocity" =====

// folder: LAxisCtrl_Blocks/InternalSubBlocks

FUNCTION "LAxisCtrl_UnpubAxisReferencingVelocity" : LReal   // FC30618, SCL
TITLE = LAxisCtrl_UnpubAxisReferencingVelocity
{ S7_Optimized_Access := 'TRUE' }
AUTHOR : tech.team.motioncontrol@siemens.com
FAMILY : AxisCtrl
VERSION : 1.1
// Support: tech.team.motioncontrol@siemens.com
   VAR_INPUT
      axis : DB_ANY;   // Axis specification
   END_VAR
   // Ret_Val : axis.Homing.ReferencingVelocity
BEGIN
   // Read axis parameter
   CASE TypeOfDB(#axis) OF
     TO_PositioningAxis:
       #LAxisCtrl_UnpubAxisReferencingVelocity := "LAxisCtrl_UnpubReferencingVelocityPosAxis"(#axis);

     TO_SynchronousAxis:
       #LAxisCtrl_UnpubAxisReferencingVelocity := "LAxisCtrl_UnpubReferencingVelocitySyncAxis"(#axis);

     ELSE
       #LAxisCtrl_UnpubAxisReferencingVelocity := 0.0;
   END_CASE;
END_FUNCTION

// ===== library: MasterCopy "LAxisCtrl_UnpubAxisSensorType" =====

// folder: LAxisCtrl_Blocks/InternalSubBlocks

FUNCTION "LAxisCtrl_UnpubAxisSensorType" : DInt   // FC30641, SCL
TITLE = LAxisCtrl_UnpubAxisSensorType
{ S7_Optimized_Access := 'TRUE' }
AUTHOR : tech.team.motioncontrol@siemens.com
FAMILY : AxisCtrl
VERSION : 1.1
// Support: tech.team.motioncontrol@siemens.com
   VAR_INPUT
      axis : DB_ANY;   // Axis specification
      index : Int;   // Index of sensor
   END_VAR
   // Ret_Val : axis.Sensor[index].Type
BEGIN
   // Read axis parameter
   CASE TypeOfDB(#axis) OF
     TO_PositioningAxis:
       #LAxisCtrl_UnpubAxisSensorType := "LAxisCtrl_UnpubSensorTypePosAxis"(axis := #axis, index := #index);

     TO_SynchronousAxis:
       #LAxisCtrl_UnpubAxisSensorType := "LAxisCtrl_UnpubSensorTypeSyncAxis"(axis := #axis, index := #index);

     ELSE
       #LAxisCtrl_UnpubAxisSensorType := 0; // Incremental
   END_CASE;
END_FUNCTION

// ===== library: MasterCopy "LAxisCtrl_UnpubAxisStatusWord" =====

// folder: LAxisCtrl_Blocks/InternalSubBlocks

FUNCTION "LAxisCtrl_UnpubAxisStatusWord" : DWord   // FC30619, SCL
TITLE = LAxisCtrl_UnpubAxisStatusWord
{ S7_Optimized_Access := 'TRUE' }
AUTHOR : tech.team.motioncontrol@siemens.com
FAMILY : AxisCtrl
VERSION : 1.1
// Support: tech.team.motioncontrol@siemens.com
   VAR_INPUT
      axis : DB_ANY;   // Axis specification
   END_VAR
   // Ret_Val : axis.StatusWord
BEGIN
   // Read axis parameter
   CASE TypeOfDB(#axis) OF
     TO_ExternalEncoder:
       #LAxisCtrl_UnpubAxisStatusWord := "LAnyAxis_UnpubStatusWordExtEncoder"(#axis);

     TO_SpeedAxis:
       #LAxisCtrl_UnpubAxisStatusWord := "LAnyAxis_UnpubStatusWordSpeedAxis"(#axis);

     TO_PositioningAxis:
       #LAxisCtrl_UnpubAxisStatusWord := "LAnyAxis_UnpubStatusWordPosAxis"(#axis);

     TO_SynchronousAxis:
       #LAxisCtrl_UnpubAxisStatusWord := "LAnyAxis_UnpubStatusWordSyncAxis"(#axis);

     ELSE
       #LAxisCtrl_UnpubAxisStatusWord := 16#0000_0000; // Invalid TO specification
   END_CASE;
END_FUNCTION

// ===== library: MasterCopy "LAxisCtrl_UnpubFunctionStateSyncAxis" =====

// folder: LAxisCtrl_Blocks/InternalSubBlocks

FUNCTION "LAxisCtrl_UnpubFunctionStateSyncAxis" : DInt   // FC30652, SCL
TITLE = LAxisCtrl_UnpubFunctionStateSyncAxis
{ S7_Optimized_Access := 'TRUE' }
AUTHOR : tech.team.motioncontrol@siemens.com
FAMILY : AxisCtrl
VERSION : 1.2
// Support: tech.team.motioncontrol@siemens.com
   VAR_INPUT
      axis : TO_SynchronousAxis;   // Axis specification
   END_VAR
   // Ret_Val : axis.StatusSynchronizedMotion.FunctionState
BEGIN
   // Read axis parameter
   #LAxisCtrl_UnpubFunctionStateSyncAxis := #axis.StatusSynchronizedMotion.FunctionState;
END_FUNCTION

// ===== library: MasterCopy "LAxisCtrl_UnpubWaitingFunctionStateSyncAxis" =====

// folder: LAxisCtrl_Blocks/InternalSubBlocks

FUNCTION "LAxisCtrl_UnpubWaitingFunctionStateSyncAxis" : DInt   // FC30639, SCL
TITLE = LAxisCtrl_UnpubWaitingFunctionStateSyncAxis
{ S7_Optimized_Access := 'TRUE' }
AUTHOR : tech.team.motioncontrol@siemens.com
FAMILY : AxisCtrl
VERSION : 1.1
// Support: tech.team.motioncontrol@siemens.com
   VAR_INPUT
      axis : TO_SynchronousAxis;   // Axis specification
   END_VAR
   // Ret_Val : axis.StatusSynchronizedMotion.WaitingFunctionState
BEGIN
   // Read axis parameter
   #LAxisCtrl_UnpubWaitingFunctionStateSyncAxis := #axis.StatusSynchronizedMotion.WaitingFunctionState;
END_FUNCTION

// ===== library: MasterCopy "LAxisCtrl_UnpubDynamicDefaultAccPosAxis" =====

// folder: LAxisCtrl_Blocks/InternalSubBlocks/DynamicDefaults

FUNCTION "LAxisCtrl_UnpubDynamicDefaultAccPosAxis" : LReal   // FC30620, SCL
TITLE = LAxisCtrl_UnpubDynamicDefaultAccPosAxis
{ S7_Optimized_Access := 'TRUE' }
AUTHOR : tech.team.motioncontrol@siemens.com
FAMILY : AxisCtrl
VERSION : 1.1
// Support: tech.team.motioncontrol@siemens.com
   VAR_INPUT
      axis : TO_PositioningAxis;   // Axis specification
   END_VAR
   // Ret_Val : axis.DynamicDefaults.Acceleration
BEGIN
   // Read axis parameter
   #LAxisCtrl_UnpubDynamicDefaultAccPosAxis := #axis.DynamicDefaults.Acceleration;
END_FUNCTION

// ===== library: MasterCopy "LAxisCtrl_UnpubDynamicDefaultAccSyncAxis" =====

// folder: LAxisCtrl_Blocks/InternalSubBlocks/DynamicDefaults

FUNCTION "LAxisCtrl_UnpubDynamicDefaultAccSyncAxis" : LReal   // FC30650, SCL
TITLE = LAxisCtrl_UnpubDynamicDefaultAccSyncAxis
{ S7_Optimized_Access := 'TRUE' }
AUTHOR : tech.team.motioncontrol@siemens.com
FAMILY : AxisCtrl
VERSION : 1.1
// Support: tech.team.motioncontrol@siemens.com
   VAR_INPUT
      axis : TO_SynchronousAxis;   // Axis specification
   END_VAR
   // Ret_Val : axis.DynamicDefaults.Acceleration
BEGIN
   // Read axis parameter
   #LAxisCtrl_UnpubDynamicDefaultAccSyncAxis := #axis.DynamicDefaults.Acceleration;
END_FUNCTION

// ===== library: MasterCopy "LAxisCtrl_UnpubDynamicDefaultDecPosAxis" =====

// folder: LAxisCtrl_Blocks/InternalSubBlocks/DynamicDefaults

FUNCTION "LAxisCtrl_UnpubDynamicDefaultDecPosAxis" : LReal   // FC30649, SCL
TITLE = LAxisCtrl_UnpubDynamicDefaultDecPosAxis
{ S7_Optimized_Access := 'TRUE' }
AUTHOR : tech.team.motioncontrol@siemens.com
FAMILY : AxisCtrl
VERSION : 1.1
// Support: tech.team.motioncontrol@siemens.com
   VAR_INPUT
      axis : TO_PositioningAxis;   // Axis specification
   END_VAR
   // Ret_Val : axis.DynamicDefaults.Deceleration
BEGIN
   // Read axis parameter
   #LAxisCtrl_UnpubDynamicDefaultDecPosAxis := #axis.DynamicDefaults.Deceleration;
END_FUNCTION

// ===== library: MasterCopy "LAxisCtrl_UnpubDynamicDefaultDecSyncAxis" =====

// folder: LAxisCtrl_Blocks/InternalSubBlocks/DynamicDefaults

FUNCTION "LAxisCtrl_UnpubDynamicDefaultDecSyncAxis" : LReal   // FC30648, SCL
TITLE = LAxisCtrl_UnpubDynamicDefaultDecSyncAxis
{ S7_Optimized_Access := 'TRUE' }
AUTHOR : tech.team.motioncontrol@siemens.com
FAMILY : AxisCtrl
VERSION : 1.1
// Support: tech.team.motioncontrol@siemens.com
   VAR_INPUT
      axis : TO_SynchronousAxis;   // Axis specification
   END_VAR
   // Ret_Val : axis.DynamicDefaults.Deceleration
BEGIN
   // Read axis parameter
   #LAxisCtrl_UnpubDynamicDefaultDecSyncAxis := #axis.DynamicDefaults.Deceleration;
END_FUNCTION

// ===== library: MasterCopy "LAxisCtrl_UnpubDynamicDefaultJerkPosAxis" =====

// folder: LAxisCtrl_Blocks/InternalSubBlocks/DynamicDefaults

FUNCTION "LAxisCtrl_UnpubDynamicDefaultJerkPosAxis" : LReal   // FC30647, SCL
TITLE = LAxisCtrl_UnpubDynamicDefaultJerkPosAxis
{ S7_Optimized_Access := 'TRUE' }
AUTHOR : tech.team.motioncontrol@siemens.com
FAMILY : AxisCtrl
VERSION : 1.1
// Support: tech.team.motioncontrol@siemens.com
   VAR_INPUT
      axis : TO_PositioningAxis;   // Axis specification
   END_VAR
   // Ret_Val : axis.DynamicDefaults.Jerk
BEGIN
   // Read axis parameter
   #LAxisCtrl_UnpubDynamicDefaultJerkPosAxis := #axis.DynamicDefaults.Jerk;
END_FUNCTION

// ===== library: MasterCopy "LAxisCtrl_UnpubDynamicDefaultJerkSyncAxis" =====

// folder: LAxisCtrl_Blocks/InternalSubBlocks/DynamicDefaults

FUNCTION "LAxisCtrl_UnpubDynamicDefaultJerkSyncAxis" : LReal   // FC30651, SCL
TITLE = LAxisCtrl_UnpubDynamicDefaultJerkSyncAxis
{ S7_Optimized_Access := 'TRUE' }
AUTHOR : tech.team.motioncontrol@siemens.com
FAMILY : AxisCtrl
VERSION : 1.1
// Support: tech.team.motioncontrol@siemens.com
   VAR_INPUT
      axis : TO_SynchronousAxis;   // Axis specification
   END_VAR
   // Ret_Val : axis.DynamicDefaults.Jerk
BEGIN
   // Read axis parameter
   #LAxisCtrl_UnpubDynamicDefaultJerkSyncAxis := #axis.DynamicDefaults.Jerk;
END_FUNCTION

// ===== library: MasterCopy "LAxisCtrl_UnpubEmergencyDecPosAxis" =====

// folder: LAxisCtrl_Blocks/InternalSubBlocks/EmergencyDeceleration

FUNCTION "LAxisCtrl_UnpubEmergencyDecPosAxis" : LReal   // FC30622, SCL
TITLE = LAxisCtrl_UnpubEmergencyDecPosAxis
{ S7_Optimized_Access := 'TRUE' }
AUTHOR : tech.team.motioncontrol@siemens.com
FAMILY : AxisCtrl
VERSION : 1.1
// Support: tech.team.motioncontrol@siemens.com
   VAR_INPUT
      axis : TO_PositioningAxis;   // Axis specification
   END_VAR
   // Ret_Val : axis.DynamicDefaults.EmergencyDeceleration
BEGIN
   // Read axis parameter
   #LAxisCtrl_UnpubEmergencyDecPosAxis := #axis.DynamicDefaults.EmergencyDeceleration;
END_FUNCTION

// ===== library: MasterCopy "LAxisCtrl_UnpubEmergencyDecSpeedAxis" =====

// folder: LAxisCtrl_Blocks/InternalSubBlocks/EmergencyDeceleration

FUNCTION "LAxisCtrl_UnpubEmergencyDecSpeedAxis" : LReal   // FC30623, SCL
TITLE = LAxisCtrl_UnpubEmergencyDecSpeedAxis
{ S7_Optimized_Access := 'TRUE' }
AUTHOR : tech.team.motioncontrol@siemens.com
FAMILY : AxisCtrl
VERSION : 1.1
// Support: tech.team.motioncontrol@siemens.com
   VAR_INPUT
      axis : TO_SpeedAxis;   // Axis specification
   END_VAR
   // Ret_Val : axis.DynamicDefaults.EmergencyDeceleration
BEGIN
   // Read axis parameter
   #LAxisCtrl_UnpubEmergencyDecSpeedAxis := #axis.DynamicDefaults.EmergencyDeceleration;
END_FUNCTION

// ===== library: MasterCopy "LAxisCtrl_UnpubEmergencyDecSyncAxis" =====

// folder: LAxisCtrl_Blocks/InternalSubBlocks/EmergencyDeceleration

FUNCTION "LAxisCtrl_UnpubEmergencyDecSyncAxis" : LReal   // FC30624, SCL
TITLE = LAxisCtrl_UnpubEmergencyDecSyncAxis
{ S7_Optimized_Access := 'TRUE' }
AUTHOR : tech.team.motioncontrol@siemens.com
FAMILY : AxisCtrl
VERSION : 1.1
// Support: tech.team.motioncontrol@siemens.com
   VAR_INPUT
      axis : TO_SynchronousAxis;   // Axis specification
   END_VAR
   // Ret_Val : axis.DynamicDefaults.EmergencyDeceleration
BEGIN
   // Read axis parameter
   #LAxisCtrl_UnpubEmergencyDecSyncAxis := #axis.DynamicDefaults.EmergencyDeceleration;
END_FUNCTION

// ===== library: MasterCopy "LAxisCtrl_UnpubHomingDirectionPosAxis" =====

// folder: LAxisCtrl_Blocks/InternalSubBlocks/HomingDirection

FUNCTION "LAxisCtrl_UnpubHomingDirectionPosAxis" : DInt   // FC30625, SCL
TITLE = LAxisCtrl_UnpubHomingDirectionPosAxis
{ S7_Optimized_Access := 'TRUE' }
AUTHOR : tech.team.motioncontrol@siemens.com
FAMILY : AxisCtrl
VERSION : 1.1
// Support: tech.team.motioncontrol@siemens.com
   VAR_INPUT
      axis : TO_PositioningAxis;   // Axis specification
      index : Int;   // Index of sensor
   END_VAR
   // Ret_Val : axis.Sensor[index].ActiveHoming.Direction
BEGIN
   // Read axis parameter
   #LAxisCtrl_UnpubHomingDirectionPosAxis := #axis.Sensor[#index].ActiveHoming.Direction;
END_FUNCTION

// ===== library: MasterCopy "LAxisCtrl_UnpubHomingDirectionSyncAxis" =====

// folder: LAxisCtrl_Blocks/InternalSubBlocks/HomingDirection

FUNCTION "LAxisCtrl_UnpubHomingDirectionSyncAxis" : DInt   // FC30645, SCL
TITLE = LAxisCtrl_UnpubHomingDirectionSyncAxis
{ S7_Optimized_Access := 'TRUE' }
AUTHOR : tech.team.motioncontrol@siemens.com
FAMILY : AxisCtrl
VERSION : 1.1
// Support: tech.team.motioncontrol@siemens.com
   VAR_INPUT
      axis : TO_SynchronousAxis;   // Axis specification
      index : Int;   // Index of sensor
   END_VAR
   // Ret_Val : axis.Sensor[index].ActiveHoming.Direction
BEGIN
   // Read axis parameter
   #LAxisCtrl_UnpubHomingDirectionSyncAxis := #axis.Sensor[#index].ActiveHoming.Direction;
END_FUNCTION

// ===== library: MasterCopy "LAxisCtrl_UnpubOperativeSensorPosAxis" =====

// folder: LAxisCtrl_Blocks/InternalSubBlocks/OperativeSensor

FUNCTION "LAxisCtrl_UnpubOperativeSensorPosAxis" : UDInt   // FC30626, SCL
TITLE = LAxisCtrl_UnpubOperativeSensorPosAxis
{ S7_Optimized_Access := 'TRUE' }
AUTHOR : tech.team.motioncontrol@siemens.com
FAMILY : AxisCtrl
VERSION : 1.1
// Support: tech.team.motioncontrol@siemens.com
   VAR_INPUT
      axis : TO_PositioningAxis;   // Axis specification
   END_VAR
   // Ret_Val : axis.OperativeSensor
BEGIN
   // Read axis parameter
   #LAxisCtrl_UnpubOperativeSensorPosAxis := #axis.OperativeSensor;
END_FUNCTION

// ===== library: MasterCopy "LAxisCtrl_UnpubOperativeSensorSyncAxis" =====

// folder: LAxisCtrl_Blocks/InternalSubBlocks/OperativeSensor

FUNCTION "LAxisCtrl_UnpubOperativeSensorSyncAxis" : UDInt   // FC30640, SCL
TITLE = LAxisCtrl_UnpubOperativeSensorSyncAxis
{ S7_Optimized_Access := 'TRUE' }
AUTHOR : tech.team.motioncontrol@siemens.com
FAMILY : AxisCtrl
VERSION : 1.1
// Support: tech.team.motioncontrol@siemens.com
   VAR_INPUT
      axis : TO_SynchronousAxis;   // Axis specification
   END_VAR
   // Ret_Val : axis.OperativeSensor
BEGIN
   // Read axis parameter
   #LAxisCtrl_UnpubOperativeSensorSyncAxis := #axis.OperativeSensor;
END_FUNCTION

// ===== library: MasterCopy "LAxisCtrl_UnpubPositioningDistancePosAxis" =====

// folder: LAxisCtrl_Blocks/InternalSubBlocks/PositioningDistance

FUNCTION "LAxisCtrl_UnpubPositioningDistancePosAxis" : LReal   // FC30628, SCL
TITLE = LAxisCtrl_UnpubPositioningDistancePosAxis
{ S7_Optimized_Access := 'TRUE' }
AUTHOR : tech.team.motioncontrol@siemens.com
FAMILY : AxisCtrl
VERSION : 1.1
// Support: tech.team.motioncontrol@siemens.com
   VAR_INPUT
      axis : TO_PositioningAxis;   // Axis specification
   END_VAR
   // Ret_Val : axis.StatusPositioning.Distance
BEGIN
   // Read axis parameter
   #LAxisCtrl_UnpubPositioningDistancePosAxis := #axis.StatusPositioning.Distance;
END_FUNCTION

// ===== library: MasterCopy "LAxisCtrl_UnpubPositioningDistanceSyncAxis" =====

// folder: LAxisCtrl_Blocks/InternalSubBlocks/PositioningDistance

FUNCTION "LAxisCtrl_UnpubPositioningDistanceSyncAxis" : LReal   // FC30629, SCL
TITLE = LAxisCtrl_UnpubPositioningDistanceSyncAxis
{ S7_Optimized_Access := 'TRUE' }
AUTHOR : tech.team.motioncontrol@siemens.com
FAMILY : AxisCtrl
VERSION : 1.1
// Support: tech.team.motioncontrol@siemens.com
   VAR_INPUT
      axis : TO_SynchronousAxis;   // Axis specification
   END_VAR
   // Ret_Val : axis.StatusPositioning.Distance
BEGIN
   // Read axis parameter
   #LAxisCtrl_UnpubPositioningDistanceSyncAxis := #axis.StatusPositioning.Distance;
END_FUNCTION

// ===== library: MasterCopy "LAxisCtrl_UnpubPositionTolerancePosAxis" =====

// folder: LAxisCtrl_Blocks/InternalSubBlocks/PositionTolerance

FUNCTION "LAxisCtrl_UnpubPositionTolerancePosAxis" : LReal   // FC30635, SCL
TITLE = LAxisCtrl_UnpubPositionTolerancePosAxis
{ S7_Optimized_Access := 'TRUE' }
AUTHOR : tech.team.motioncontrol@siemens.com
FAMILY : AxisCtrl
VERSION : 1.1
// Support: tech.team.motioncontrol@siemens.com
   VAR_INPUT
      axis : TO_PositioningAxis;   // Axis specification
   END_VAR
   // Ret_Val : axis.Clamping.PositionTolerance
BEGIN
   // Read axis parameter
   #LAxisCtrl_UnpubPositionTolerancePosAxis := #axis.Clamping.PositionTolerance;
END_FUNCTION

// ===== library: MasterCopy "LAxisCtrl_UnpubPositionToleranceSyncAxis" =====

// folder: LAxisCtrl_Blocks/InternalSubBlocks/PositionTolerance

FUNCTION "LAxisCtrl_UnpubPositionToleranceSyncAxis" : LReal   // FC30636, SCL
TITLE = LAxisCtrl_UnpubPositionToleranceSyncAxis
{ S7_Optimized_Access := 'TRUE' }
AUTHOR : tech.team.motioncontrol@siemens.com
FAMILY : AxisCtrl
VERSION : 1.1
// Support: tech.team.motioncontrol@siemens.com
   VAR_INPUT
      axis : TO_SynchronousAxis;   // Axis specification
   END_VAR
   // Ret_Val : axis.Clamping.PositionTolerance
BEGIN
   // Read axis parameter
   #LAxisCtrl_UnpubPositionToleranceSyncAxis := #axis.Clamping.PositionTolerance;
END_FUNCTION

// ===== library: MasterCopy "LAxisCtrl_UnpubReferencingVelocityPosAxis" =====

// folder: LAxisCtrl_Blocks/InternalSubBlocks/ReferencingVelocity

FUNCTION "LAxisCtrl_UnpubReferencingVelocityPosAxis" : LReal   // FC30637, SCL
TITLE = LAxisCtrl_UnpubReferencingVelocityPosAxis
{ S7_Optimized_Access := 'TRUE' }
AUTHOR : tech.team.motioncontrol@siemens.com
FAMILY : AxisCtrl
VERSION : 1.1
// Support: tech.team.motioncontrol@siemens.com
   VAR_INPUT
      axis : TO_PositioningAxis;   // Axis specification
   END_VAR
   // Ret_Val : axis.Homing.ReferencingVelocity
BEGIN
   // Read axis parameter
   #LAxisCtrl_UnpubReferencingVelocityPosAxis := #axis.Homing.ReferencingVelocity;
END_FUNCTION

// ===== library: MasterCopy "LAxisCtrl_UnpubReferencingVelocitySyncAxis" =====

// folder: LAxisCtrl_Blocks/InternalSubBlocks/ReferencingVelocity

